REGION Network 18: Robot1Grip Code
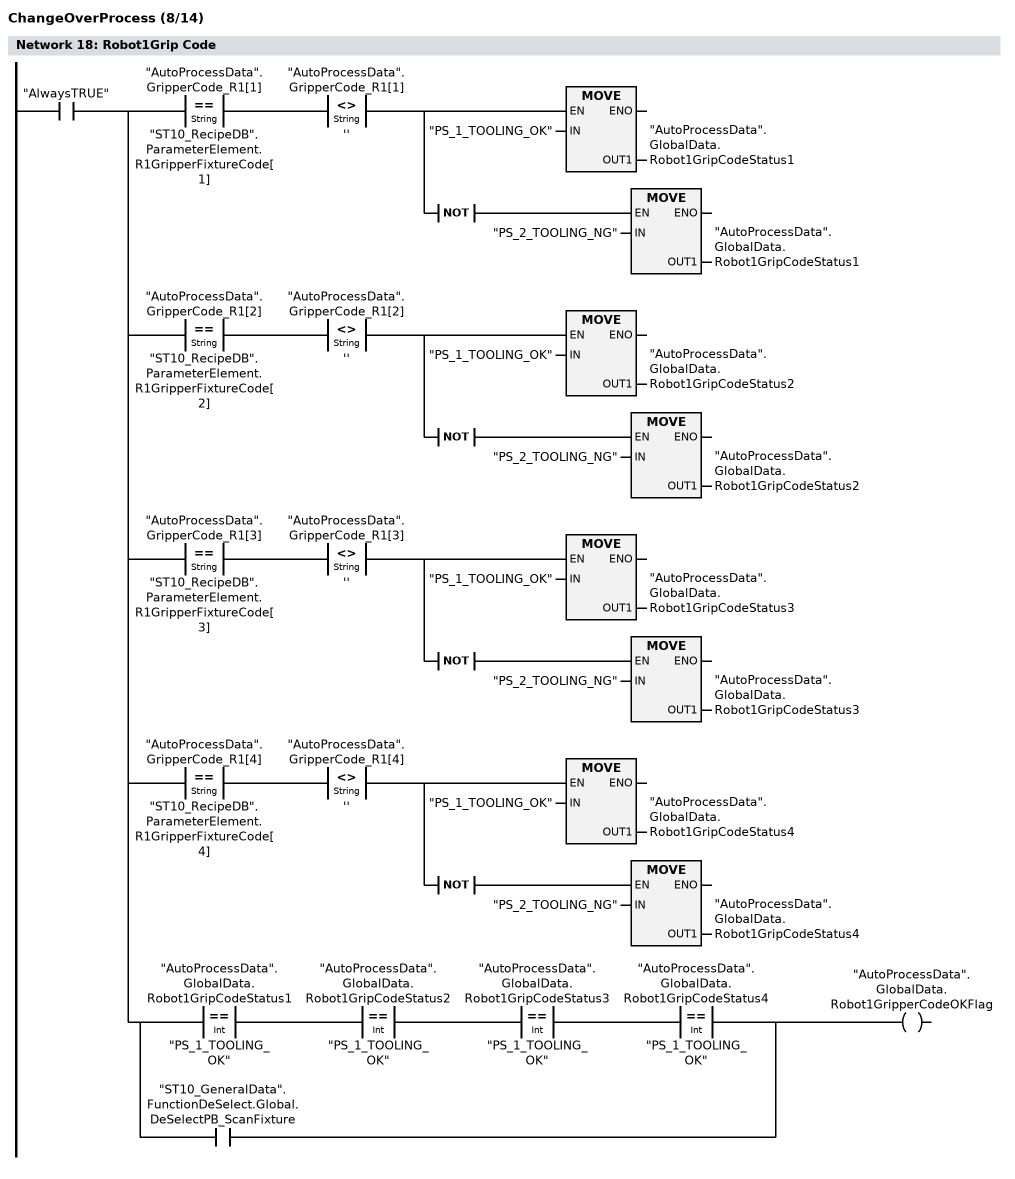
   RUNG wire#powerrail
      Contact( "AlwaysTRUE" )
      wire#w1
      { S7_Templates := "SrcType := String" } EQ_Contact(in1 := "AutoProcessData".GripperCode_R1[1], in2 := "ST10_RecipeDB".ParameterElement.R1GripperFixtureCode[1])
      { S7_Templates := "SrcType := String" } NE_Contact(in1 := "AutoProcessData".GripperCode_R1[1], in2 := '')
      wire#w2
      Move(in := "PS_1_TOOLING_OK", out1 => "AutoProcessData".GlobalData.Robot1GripCodeStatus1)
   END_RUNG
   RUNG wire#w2
      Not()
      Move(in := "PS_2_TOOLING_NG", out1 => "AutoProcessData".GlobalData.Robot1GripCodeStatus1)
   END_RUNG
   RUNG wire#w1
      { S7_Templates := "SrcType := String" } EQ_Contact(in1 := "AutoProcessData".GripperCode_R1[2], in2 := "ST10_RecipeDB".ParameterElement.R1GripperFixtureCode[2])
      { S7_Templates := "SrcType := String" } NE_Contact(in1 := "AutoProcessData".GripperCode_R1[2], in2 := '')
      wire#w3
      Move(in := "PS_1_TOOLING_OK", out1 => "AutoProcessData".GlobalData.Robot1GripCodeStatus2)
   END_RUNG
   RUNG wire#w3
      Not()
      Move(in := "PS_2_TOOLING_NG", out1 => "AutoProcessData".GlobalData.Robot1GripCodeStatus2)
   END_RUNG
   RUNG wire#w1
      { S7_Templates := "SrcType := String" } EQ_Contact(in1 := "AutoProcessData".GripperCode_R1[3], in2 := "ST10_RecipeDB".ParameterElement.R1GripperFixtureCode[3])
      { S7_Templates := "SrcType := String" } NE_Contact(in1 := "AutoProcessData".GripperCode_R1[3], in2 := '')
      wire#w4
      Move(in := "PS_1_TOOLING_OK", out1 => "AutoProcessData".GlobalData.Robot1GripCodeStatus3)
   END_RUNG
   RUNG wire#w4
      Not()
      Move(in := "PS_2_TOOLING_NG", out1 => "AutoProcessData".GlobalData.Robot1GripCodeStatus3)
   END_RUNG
   RUNG wire#w1
      { S7_Templates := "SrcType := String" } EQ_Contact(in1 := "AutoProcessData".GripperCode_R1[4], in2 := "ST10_RecipeDB".ParameterElement.R1GripperFixtureCode[4])
      { S7_Templates := "SrcType := String" } NE_Contact(in1 := "AutoProcessData".GripperCode_R1[4], in2 := '')
      wire#w5
      Move(in := "PS_1_TOOLING_OK", out1 => "AutoProcessData".GlobalData.Robot1GripCodeStatus4)
   END_RUNG
   RUNG wire#w5
      Not()
      Move(in := "PS_2_TOOLING_NG", out1 => "AutoProcessData".GlobalData.Robot1GripCodeStatus4)
   END_RUNG
   RUNG wire#w1
      { S7_Templates := "SrcType := Int" } EQ_Contact(in1 := "AutoProcessData".GlobalData.Robot1GripCodeStatus1, in2 := "PS_1_TOOLING_OK")
      { S7_Templates := "SrcType := Int" } EQ_Contact(in1 := "AutoProcessData".GlobalData.Robot1GripCodeStatus2, in2 := "PS_1_TOOLING_OK")
      { S7_Templates := "SrcType := Int" } EQ_Contact(in1 := "AutoProcessData".GlobalData.Robot1GripCodeStatus3, in2 := "PS_1_TOOLING_OK")
      { S7_Templates := "SrcType := Int" } EQ_Contact(in1 := "AutoProcessData".GlobalData.Robot1GripCodeStatus4, in2 := "PS_1_TOOLING_OK")
      wire#w6
      Coil( "AutoProcessData".GlobalData.Robot1GripperCodeOKFlag )
   END_RUNG
   RUNG wire#w1
      Contact( "ST10_GeneralData".FunctionDeSelect.Global.DeSelectPB_ScanFixture )
   END_RUNG wire#w6
   // the same network as SCL:
   #_w1 := "AlwaysTRUE" AND ("AutoProcessData".GripperCode_R1[1] = "ST10_RecipeDB".ParameterElement.R1GripperFixtureCode[1]) AND ("AutoProcessData".GripperCode_R1[1] <> '');
   IF #_w1 THEN "AutoProcessData".GlobalData.Robot1GripCodeStatus1 := "PS_1_TOOLING_OK"; END_IF;
   IF NOT #_w1 THEN "AutoProcessData".GlobalData.Robot1GripCodeStatus1 := "PS_2_TOOLING_NG"; END_IF;
   #_w2 := "AlwaysTRUE" AND ("AutoProcessData".GripperCode_R1[2] = "ST10_RecipeDB".ParameterElement.R1GripperFixtureCode[2]) AND ("AutoProcessData".GripperCode_R1[2] <> '');
   IF #_w2 THEN "AutoProcessData".GlobalData.Robot1GripCodeStatus2 := "PS_1_TOOLING_OK"; END_IF;
   IF NOT #_w2 THEN "AutoProcessData".GlobalData.Robot1GripCodeStatus2 := "PS_2_TOOLING_NG"; END_IF;
   #_w3 := "AlwaysTRUE" AND ("AutoProcessData".GripperCode_R1[3] = "ST10_RecipeDB".ParameterElement.R1GripperFixtureCode[3]) AND ("AutoProcessData".GripperCode_R1[3] <> '');
   IF #_w3 THEN "AutoProcessData".GlobalData.Robot1GripCodeStatus3 := "PS_1_TOOLING_OK"; END_IF;
   IF NOT #_w3 THEN "AutoProcessData".GlobalData.Robot1GripCodeStatus3 := "PS_2_TOOLING_NG"; END_IF;
   #_w4 := "AlwaysTRUE" AND ("AutoProcessData".GripperCode_R1[4] = "ST10_RecipeDB".ParameterElement.R1GripperFixtureCode[4]) AND ("AutoProcessData".GripperCode_R1[4] <> '');
   IF #_w4 THEN "AutoProcessData".GlobalData.Robot1GripCodeStatus4 := "PS_1_TOOLING_OK"; END_IF;
   IF NOT #_w4 THEN "AutoProcessData".GlobalData.Robot1GripCodeStatus4 := "PS_2_TOOLING_NG"; END_IF;
   "AutoProcessData".GlobalData.Robot1GripperCodeOKFlag := "AlwaysTRUE" AND ((("AutoProcessData".GlobalData.Robot1GripCodeStatus1 = "PS_1_TOOLING_OK") AND ("AutoProcessData".GlobalData.Robot1GripCodeStatus2 = "PS_1_TOOLING_OK") AND ("AutoProcessData".GlobalData.Robot1GripCodeStatus3 = "PS_1_TOOLING_OK") AND ("AutoProcessData".GlobalData.Robot1GripCodeStatus4 = "PS_1_TOOLING_OK")) OR "ST10_GeneralData".FunctionDeSelect.Global.DeSelectPB_ScanFixture);
END_REGION

REGION Network 19: Robot2Grip Code
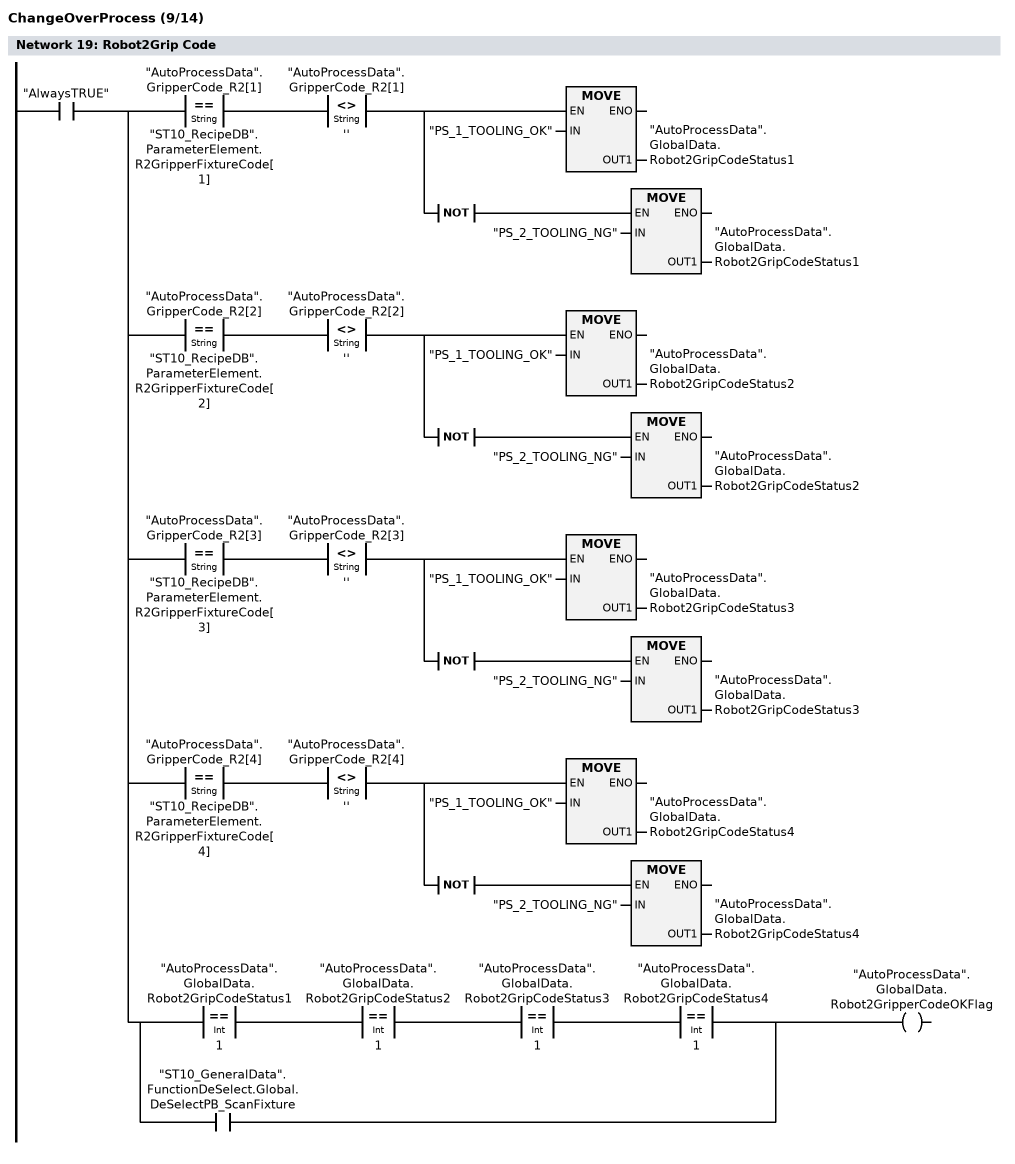
   RUNG wire#powerrail
      Contact( "AlwaysTRUE" )
      wire#w1
      { S7_Templates := "SrcType := String" } EQ_Contact(in1 := "AutoProcessData".GripperCode_R2[1], in2 := "ST10_RecipeDB".ParameterElement.R2GripperFixtureCode[1])
      { S7_Templates := "SrcType := String" } NE_Contact(in1 := "AutoProcessData".GripperCode_R2[1], in2 := '')
      wire#w2
      Move(in := "PS_1_TOOLING_OK", out1 => "AutoProcessData".GlobalData.Robot2GripCodeStatus1)
   END_RUNG
   RUNG wire#w2
      Not()
      Move(in := "PS_2_TOOLING_NG", out1 => "AutoProcessData".GlobalData.Robot2GripCodeStatus1)
   END_RUNG
   RUNG wire#w1
      { S7_Templates := "SrcType := String" } EQ_Contact(in1 := "AutoProcessData".GripperCode_R2[2], in2 := "ST10_RecipeDB".ParameterElement.R2GripperFixtureCode[2])
      { S7_Templates := "SrcType := String" } NE_Contact(in1 := "AutoProcessData".GripperCode_R2[2], in2 := '')
      wire#w3
      Move(in := "PS_1_TOOLING_OK", out1 => "AutoProcessData".GlobalData.Robot2GripCodeStatus2)
   END_RUNG
   RUNG wire#w3
      Not()
      Move(in := "PS_2_TOOLING_NG", out1 => "AutoProcessData".GlobalData.Robot2GripCodeStatus2)
   END_RUNG
   RUNG wire#w1
      { S7_Templates := "SrcType := String" } EQ_Contact(in1 := "AutoProcessData".GripperCode_R2[3], in2 := "ST10_RecipeDB".ParameterElement.R2GripperFixtureCode[3])
      { S7_Templates := "SrcType := String" } NE_Contact(in1 := "AutoProcessData".GripperCode_R2[3], in2 := '')
      wire#w4
      Move(in := "PS_1_TOOLING_OK", out1 => "AutoProcessData".GlobalData.Robot2GripCodeStatus3)
   END_RUNG
   RUNG wire#w4
      Not()
      Move(in := "PS_2_TOOLING_NG", out1 => "AutoProcessData".GlobalData.Robot2GripCodeStatus3)
   END_RUNG
   RUNG wire#w1
      { S7_Templates := "SrcType := String" } EQ_Contact(in1 := "AutoProcessData".GripperCode_R2[4], in2 := "ST10_RecipeDB".ParameterElement.R2GripperFixtureCode[4])
      { S7_Templates := "SrcType := String" } NE_Contact(in1 := "AutoProcessData".GripperCode_R2[4], in2 := '')
      wire#w5
      Move(in := "PS_1_TOOLING_OK", out1 => "AutoProcessData".GlobalData.Robot2GripCodeStatus4)
   END_RUNG
   RUNG wire#w5
      Not()
      Move(in := "PS_2_TOOLING_NG", out1 => "AutoProcessData".GlobalData.Robot2GripCodeStatus4)
   END_RUNG
   RUNG wire#w1
      { S7_Templates := "SrcType := Int" } EQ_Contact(in1 := "AutoProcessData".GlobalData.Robot2GripCodeStatus1, in2 := 1)
      { S7_Templates := "SrcType := Int" } EQ_Contact(in1 := "AutoProcessData".GlobalData.Robot2GripCodeStatus2, in2 := 1)
      { S7_Templates := "SrcType := Int" } EQ_Contact(in1 := "AutoProcessData".GlobalData.Robot2GripCodeStatus3, in2 := 1)
      { S7_Templates := "SrcType := Int" } EQ_Contact(in1 := "AutoProcessData".GlobalData.Robot2GripCodeStatus4, in2 := 1)
      wire#w6
      Coil( "AutoProcessData".GlobalData.Robot2GripperCodeOKFlag )
   END_RUNG
   RUNG wire#w1
      Contact( "ST10_GeneralData".FunctionDeSelect.Global.DeSelectPB_ScanFixture )
   END_RUNG wire#w6
   // the same network as SCL:
   #_w1 := "AlwaysTRUE" AND ("AutoProcessData".GripperCode_R2[1] = "ST10_RecipeDB".ParameterElement.R2GripperFixtureCode[1]) AND ("AutoProcessData".GripperCode_R2[1] <> '');
   IF #_w1 THEN "AutoProcessData".GlobalData.Robot2GripCodeStatus1 := "PS_1_TOOLING_OK"; END_IF;
   IF NOT #_w1 THEN "AutoProcessData".GlobalData.Robot2GripCodeStatus1 := "PS_2_TOOLING_NG"; END_IF;
   #_w2 := "AlwaysTRUE" AND ("AutoProcessData".GripperCode_R2[2] = "ST10_RecipeDB".ParameterElement.R2GripperFixtureCode[2]) AND ("AutoProcessData".GripperCode_R2[2] <> '');
   IF #_w2 THEN "AutoProcessData".GlobalData.Robot2GripCodeStatus2 := "PS_1_TOOLING_OK"; END_IF;
   IF NOT #_w2 THEN "AutoProcessData".GlobalData.Robot2GripCodeStatus2 := "PS_2_TOOLING_NG"; END_IF;
   #_w3 := "AlwaysTRUE" AND ("AutoProcessData".GripperCode_R2[3] = "ST10_RecipeDB".ParameterElement.R2GripperFixtureCode[3]) AND ("AutoProcessData".GripperCode_R2[3] <> '');
   IF #_w3 THEN "AutoProcessData".GlobalData.Robot2GripCodeStatus3 := "PS_1_TOOLING_OK"; END_IF;
   IF NOT #_w3 THEN "AutoProcessData".GlobalData.Robot2GripCodeStatus3 := "PS_2_TOOLING_NG"; END_IF;
   #_w4 := "AlwaysTRUE" AND ("AutoProcessData".GripperCode_R2[4] = "ST10_RecipeDB".ParameterElement.R2GripperFixtureCode[4]) AND ("AutoProcessData".GripperCode_R2[4] <> '');
   IF #_w4 THEN "AutoProcessData".GlobalData.Robot2GripCodeStatus4 := "PS_1_TOOLING_OK"; END_IF;
   IF NOT #_w4 THEN "AutoProcessData".GlobalData.Robot2GripCodeStatus4 := "PS_2_TOOLING_NG"; END_IF;
   "AutoProcessData".GlobalData.Robot2GripperCodeOKFlag := "AlwaysTRUE" AND ((("AutoProcessData".GlobalData.Robot2GripCodeStatus1 = 1) AND ("AutoProcessData".GlobalData.Robot2GripCodeStatus2 = 1) AND ("AutoProcessData".GlobalData.Robot2GripCodeStatus3 = 1) AND ("AutoProcessData".GlobalData.Robot2GripCodeStatus4 = 1)) OR "ST10_GeneralData".FunctionDeSelect.Global.DeSelectPB_ScanFixture);
END_REGION

REGION Network 20: Robot3Grip Code
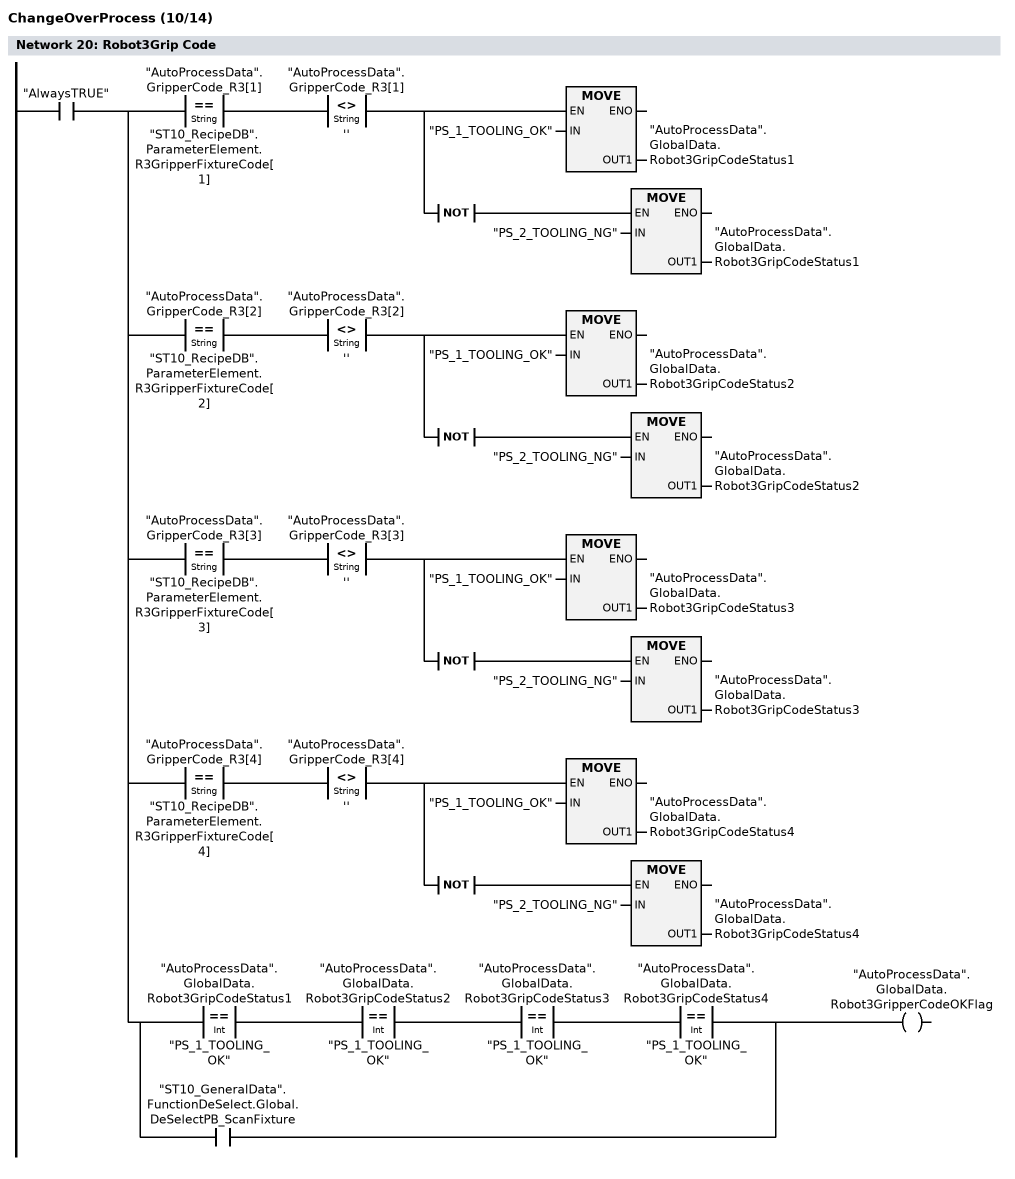
   RUNG wire#powerrail
      Contact( "AlwaysTRUE" )
      wire#w1
      { S7_Templates := "SrcType := String" } EQ_Contact(in1 := "AutoProcessData".GripperCode_R3[1], in2 := "ST10_RecipeDB".ParameterElement.R3GripperFixtureCode[1])
      { S7_Templates := "SrcType := String" } NE_Contact(in1 := "AutoProcessData".GripperCode_R3[1], in2 := '')
      wire#w2
      Move(in := "PS_1_TOOLING_OK", out1 => "AutoProcessData".GlobalData.Robot3GripCodeStatus1)
   END_RUNG
   RUNG wire#w2
      Not()
      Move(in := "PS_2_TOOLING_NG", out1 => "AutoProcessData".GlobalData.Robot3GripCodeStatus1)
   END_RUNG
   RUNG wire#w1
      { S7_Templates := "SrcType := String" } EQ_Contact(in1 := "AutoProcessData".GripperCode_R3[2], in2 := "ST10_RecipeDB".ParameterElement.R3GripperFixtureCode[2])
      { S7_Templates := "SrcType := String" } NE_Contact(in1 := "AutoProcessData".GripperCode_R3[2], in2 := '')
      wire#w3
      Move(in := "PS_1_TOOLING_OK", out1 => "AutoProcessData".GlobalData.Robot3GripCodeStatus2)
   END_RUNG
   RUNG wire#w3
      Not()
      Move(in := "PS_2_TOOLING_NG", out1 => "AutoProcessData".GlobalData.Robot3GripCodeStatus2)
   END_RUNG
   RUNG wire#w1
      { S7_Templates := "SrcType := String" } EQ_Contact(in1 := "AutoProcessData".GripperCode_R3[3], in2 := "ST10_RecipeDB".ParameterElement.R3GripperFixtureCode[3])
      { S7_Templates := "SrcType := String" } NE_Contact(in1 := "AutoProcessData".GripperCode_R3[3], in2 := '')
      wire#w4
      Move(in := "PS_1_TOOLING_OK", out1 => "AutoProcessData".GlobalData.Robot3GripCodeStatus3)
   END_RUNG
   RUNG wire#w4
      Not()
      Move(in := "PS_2_TOOLING_NG", out1 => "AutoProcessData".GlobalData.Robot3GripCodeStatus3)
   END_RUNG
   RUNG wire#w1
      { S7_Templates := "SrcType := String" } EQ_Contact(in1 := "AutoProcessData".GripperCode_R3[4], in2 := "ST10_RecipeDB".ParameterElement.R3GripperFixtureCode[4])
      { S7_Templates := "SrcType := String" } NE_Contact(in1 := "AutoProcessData".GripperCode_R3[4], in2 := '')
      wire#w5
      Move(in := "PS_1_TOOLING_OK", out1 => "AutoProcessData".GlobalData.Robot3GripCodeStatus4)
   END_RUNG
   RUNG wire#w5
      Not()
      Move(in := "PS_2_TOOLING_NG", out1 => "AutoProcessData".GlobalData.Robot3GripCodeStatus4)
   END_RUNG
   RUNG wire#w1
      { S7_Templates := "SrcType := Int" } EQ_Contact(in1 := "AutoProcessData".GlobalData.Robot3GripCodeStatus1, in2 := "PS_1_TOOLING_OK")
      { S7_Templates := "SrcType := Int" } EQ_Contact(in1 := "AutoProcessData".GlobalData.Robot3GripCodeStatus2, in2 := "PS_1_TOOLING_OK")
      { S7_Templates := "SrcType := Int" } EQ_Contact(in1 := "AutoProcessData".GlobalData.Robot3GripCodeStatus3, in2 := "PS_1_TOOLING_OK")
      { S7_Templates := "SrcType := Int" } EQ_Contact(in1 := "AutoProcessData".GlobalData.Robot3GripCodeStatus4, in2 := "PS_1_TOOLING_OK")
      wire#w6
      Coil( "AutoProcessData".GlobalData.Robot3GripperCodeOKFlag )
   END_RUNG
   RUNG wire#w1
      Contact( "ST10_GeneralData".FunctionDeSelect.Global.DeSelectPB_ScanFixture )
   END_RUNG wire#w6
   // the same network as SCL:
   #_w1 := "AlwaysTRUE" AND ("AutoProcessData".GripperCode_R3[1] = "ST10_RecipeDB".ParameterElement.R3GripperFixtureCode[1]) AND ("AutoProcessData".GripperCode_R3[1] <> '');
   IF #_w1 THEN "AutoProcessData".GlobalData.Robot3GripCodeStatus1 := "PS_1_TOOLING_OK"; END_IF;
   IF NOT #_w1 THEN "AutoProcessData".GlobalData.Robot3GripCodeStatus1 := "PS_2_TOOLING_NG"; END_IF;
   #_w2 := "AlwaysTRUE" AND ("AutoProcessData".GripperCode_R3[2] = "ST10_RecipeDB".ParameterElement.R3GripperFixtureCode[2]) AND ("AutoProcessData".GripperCode_R3[2] <> '');
   IF #_w2 THEN "AutoProcessData".GlobalData.Robot3GripCodeStatus2 := "PS_1_TOOLING_OK"; END_IF;
   IF NOT #_w2 THEN "AutoProcessData".GlobalData.Robot3GripCodeStatus2 := "PS_2_TOOLING_NG"; END_IF;
   #_w3 := "AlwaysTRUE" AND ("AutoProcessData".GripperCode_R3[3] = "ST10_RecipeDB".ParameterElement.R3GripperFixtureCode[3]) AND ("AutoProcessData".GripperCode_R3[3] <> '');
   IF #_w3 THEN "AutoProcessData".GlobalData.Robot3GripCodeStatus3 := "PS_1_TOOLING_OK"; END_IF;
   IF NOT #_w3 THEN "AutoProcessData".GlobalData.Robot3GripCodeStatus3 := "PS_2_TOOLING_NG"; END_IF;
   #_w4 := "AlwaysTRUE" AND ("AutoProcessData".GripperCode_R3[4] = "ST10_RecipeDB".ParameterElement.R3GripperFixtureCode[4]) AND ("AutoProcessData".GripperCode_R3[4] <> '');
   IF #_w4 THEN "AutoProcessData".GlobalData.Robot3GripCodeStatus4 := "PS_1_TOOLING_OK"; END_IF;
   IF NOT #_w4 THEN "AutoProcessData".GlobalData.Robot3GripCodeStatus4 := "PS_2_TOOLING_NG"; END_IF;
   "AutoProcessData".GlobalData.Robot3GripperCodeOKFlag := "AlwaysTRUE" AND ((("AutoProcessData".GlobalData.Robot3GripCodeStatus1 = "PS_1_TOOLING_OK") AND ("AutoProcessData".GlobalData.Robot3GripCodeStatus2 = "PS_1_TOOLING_OK") AND ("AutoProcessData".GlobalData.Robot3GripCodeStatus3 = "PS_1_TOOLING_OK") AND ("AutoProcessData".GlobalData.Robot3GripCodeStatus4 = "PS_1_TOOLING_OK")) OR "ST10_GeneralData".FunctionDeSelect.Global.DeSelectPB_ScanFixture);
END_REGION

REGION Network 21: A1 Fixture Code
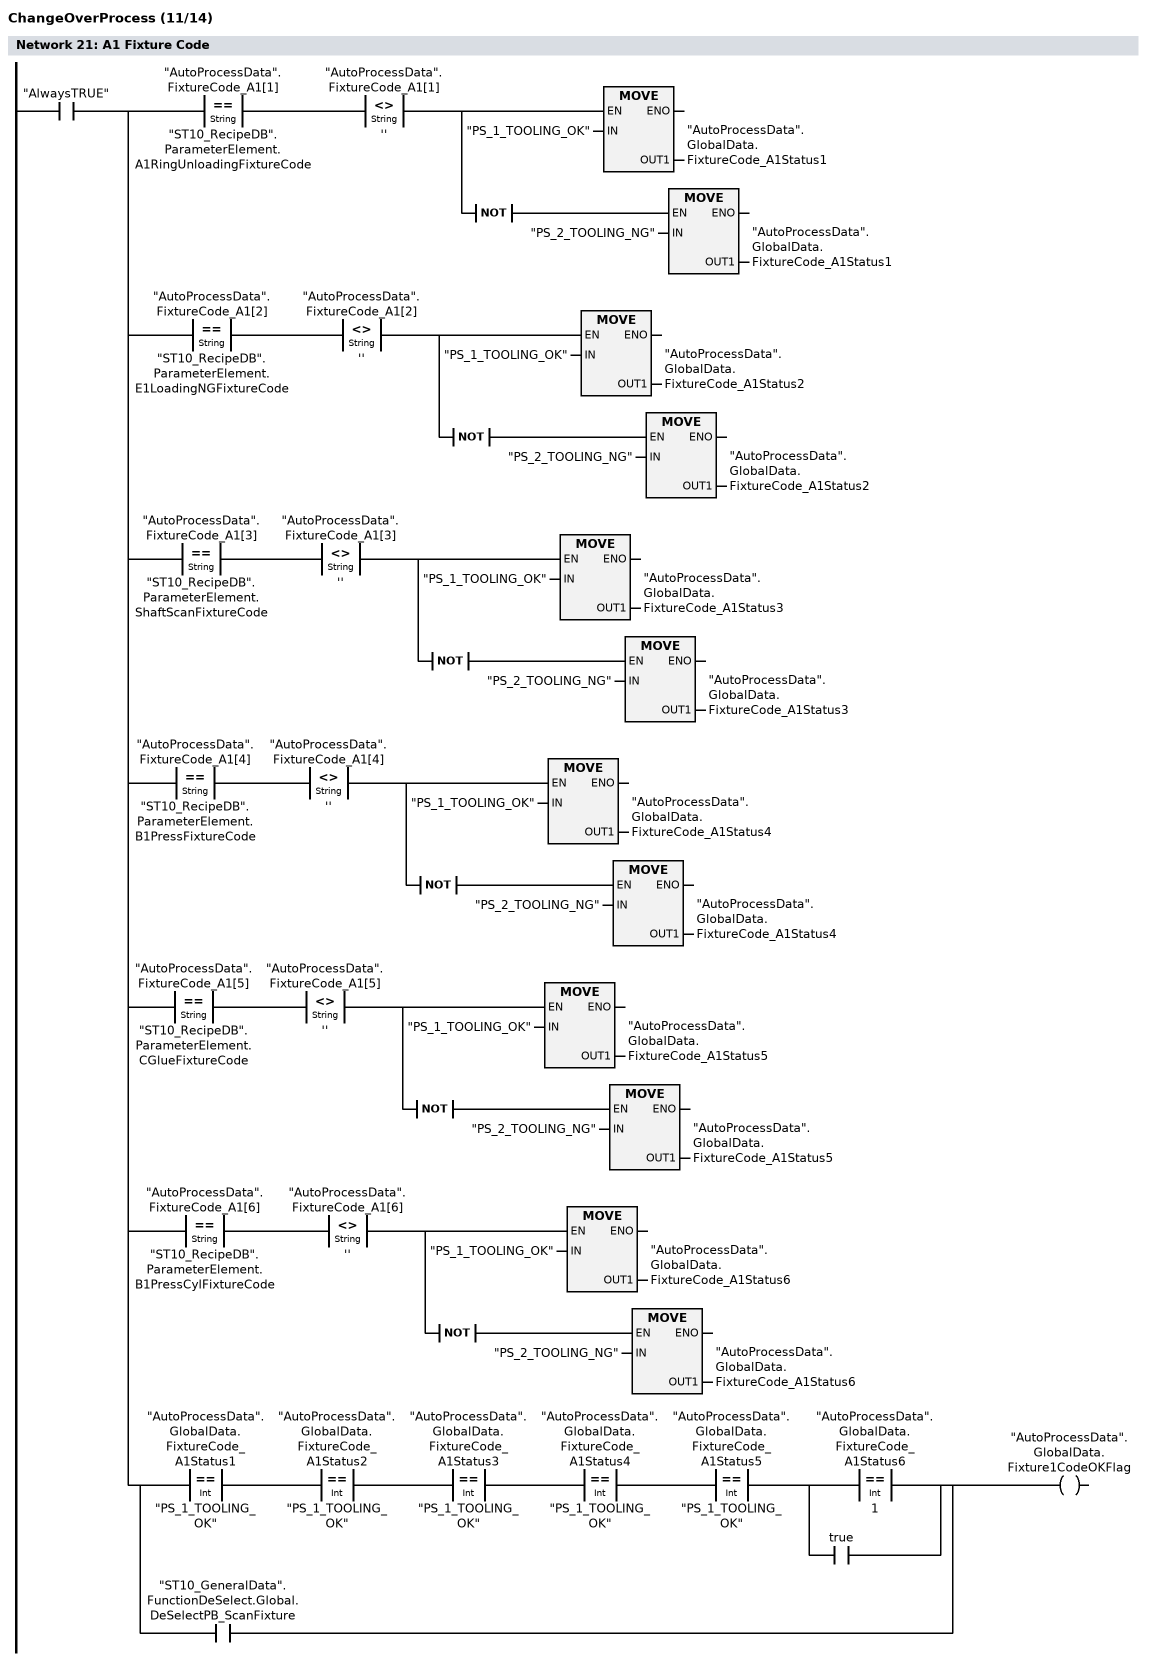
   RUNG wire#powerrail
      Contact( "AlwaysTRUE" )
      wire#w1
      { S7_Templates := "SrcType := String" } EQ_Contact(in1 := "AutoProcessData".FixtureCode_A1[1], in2 := "ST10_RecipeDB".ParameterElement.A1RingUnloadingFixtureCode)
      { S7_Templates := "SrcType := String" } NE_Contact(in1 := "AutoProcessData".FixtureCode_A1[1], in2 := '')
      wire#w2
      Move(in := "PS_1_TOOLING_OK", out1 => "AutoProcessData".GlobalData.FixtureCode_A1Status1)
   END_RUNG
   RUNG wire#w2
      Not()
      Move(in := "PS_2_TOOLING_NG", out1 => "AutoProcessData".GlobalData.FixtureCode_A1Status1)
   END_RUNG
   RUNG wire#w1
      { S7_Templates := "SrcType := String" } EQ_Contact(in1 := "AutoProcessData".FixtureCode_A1[2], in2 := "ST10_RecipeDB".ParameterElement.E1LoadingNGFixtureCode)
      { S7_Templates := "SrcType := String" } NE_Contact(in1 := "AutoProcessData".FixtureCode_A1[2], in2 := '')
      wire#w3
      Move(in := "PS_1_TOOLING_OK", out1 => "AutoProcessData".GlobalData.FixtureCode_A1Status2)
   END_RUNG
   RUNG wire#w3
      Not()
      Move(in := "PS_2_TOOLING_NG", out1 => "AutoProcessData".GlobalData.FixtureCode_A1Status2)
   END_RUNG
   RUNG wire#w1
      { S7_Templates := "SrcType := String" } EQ_Contact(in1 := "AutoProcessData".FixtureCode_A1[3], in2 := "ST10_RecipeDB".ParameterElement.ShaftScanFixtureCode)
      { S7_Templates := "SrcType := String" } NE_Contact(in1 := "AutoProcessData".FixtureCode_A1[3], in2 := '')
      wire#w4
      Move(in := "PS_1_TOOLING_OK", out1 => "AutoProcessData".GlobalData.FixtureCode_A1Status3)
   END_RUNG
   RUNG wire#w4
      Not()
      Move(in := "PS_2_TOOLING_NG", out1 => "AutoProcessData".GlobalData.FixtureCode_A1Status3)
   END_RUNG
   RUNG wire#w1
      { S7_Templates := "SrcType := String" } EQ_Contact(in1 := "AutoProcessData".FixtureCode_A1[4], in2 := "ST10_RecipeDB".ParameterElement.B1PressFixtureCode)
      { S7_Templates := "SrcType := String" } NE_Contact(in1 := "AutoProcessData".FixtureCode_A1[4], in2 := '')
      wire#w5
      Move(in := "PS_1_TOOLING_OK", out1 => "AutoProcessData".GlobalData.FixtureCode_A1Status4)
   END_RUNG
   RUNG wire#w5
      Not()
      Move(in := "PS_2_TOOLING_NG", out1 => "AutoProcessData".GlobalData.FixtureCode_A1Status4)
   END_RUNG
   RUNG wire#w1
      { S7_Templates := "SrcType := String" } EQ_Contact(in1 := "AutoProcessData".FixtureCode_A1[5], in2 := "ST10_RecipeDB".ParameterElement.CGlueFixtureCode)
      { S7_Templates := "SrcType := String" } NE_Contact(in1 := "AutoProcessData".FixtureCode_A1[5], in2 := '')
      wire#w6
      Move(in := "PS_1_TOOLING_OK", out1 => "AutoProcessData".GlobalData.FixtureCode_A1Status5)
   END_RUNG
   RUNG wire#w6
      Not()
      Move(in := "PS_2_TOOLING_NG", out1 => "AutoProcessData".GlobalData.FixtureCode_A1Status5)
   END_RUNG
   RUNG wire#w1
      { S7_Templates := "SrcType := String" } EQ_Contact(in1 := "AutoProcessData".FixtureCode_A1[6], in2 := "ST10_RecipeDB".ParameterElement.B1PressCylFixtureCode)
      { S7_Templates := "SrcType := String" } NE_Contact(in1 := "AutoProcessData".FixtureCode_A1[6], in2 := '')
      wire#w7
      Move(in := "PS_1_TOOLING_OK", out1 => "AutoProcessData".GlobalData.FixtureCode_A1Status6)
   END_RUNG
   RUNG wire#w7
      Not()
      Move(in := "PS_2_TOOLING_NG", out1 => "AutoProcessData".GlobalData.FixtureCode_A1Status6)
   END_RUNG
   RUNG wire#w1
      { S7_Templates := "SrcType := Int" } EQ_Contact(in1 := "AutoProcessData".GlobalData.FixtureCode_A1Status1, in2 := "PS_1_TOOLING_OK")
      { S7_Templates := "SrcType := Int" } EQ_Contact(in1 := "AutoProcessData".GlobalData.FixtureCode_A1Status2, in2 := "PS_1_TOOLING_OK")
      { S7_Templates := "SrcType := Int" } EQ_Contact(in1 := "AutoProcessData".GlobalData.FixtureCode_A1Status3, in2 := "PS_1_TOOLING_OK")
      { S7_Templates := "SrcType := Int" } EQ_Contact(in1 := "AutoProcessData".GlobalData.FixtureCode_A1Status4, in2 := "PS_1_TOOLING_OK")
      { S7_Templates := "SrcType := Int" } EQ_Contact(in1 := "AutoProcessData".GlobalData.FixtureCode_A1Status5, in2 := "PS_1_TOOLING_OK")
      wire#w8
      { S7_Templates := "SrcType := Int" } EQ_Contact(in1 := "AutoProcessData".GlobalData.FixtureCode_A1Status6, in2 := 1)
      wire#w9
      Coil( "AutoProcessData".GlobalData.Fixture1CodeOKFlag )
   END_RUNG
   RUNG wire#w8
      Contact( true )
   END_RUNG wire#w9
   RUNG wire#w1
      Contact( "ST10_GeneralData".FunctionDeSelect.Global.DeSelectPB_ScanFixture )
   END_RUNG wire#w9
   // the same network as SCL:
   #_w1 := "AlwaysTRUE" AND ("AutoProcessData".FixtureCode_A1[1] = "ST10_RecipeDB".ParameterElement.A1RingUnloadingFixtureCode) AND ("AutoProcessData".FixtureCode_A1[1] <> '');
   IF #_w1 THEN "AutoProcessData".GlobalData.FixtureCode_A1Status1 := "PS_1_TOOLING_OK"; END_IF;
   IF NOT #_w1 THEN "AutoProcessData".GlobalData.FixtureCode_A1Status1 := "PS_2_TOOLING_NG"; END_IF;
   #_w2 := "AlwaysTRUE" AND ("AutoProcessData".FixtureCode_A1[2] = "ST10_RecipeDB".ParameterElement.E1LoadingNGFixtureCode) AND ("AutoProcessData".FixtureCode_A1[2] <> '');
   IF #_w2 THEN "AutoProcessData".GlobalData.FixtureCode_A1Status2 := "PS_1_TOOLING_OK"; END_IF;
   IF NOT #_w2 THEN "AutoProcessData".GlobalData.FixtureCode_A1Status2 := "PS_2_TOOLING_NG"; END_IF;
   #_w3 := "AlwaysTRUE" AND ("AutoProcessData".FixtureCode_A1[3] = "ST10_RecipeDB".ParameterElement.ShaftScanFixtureCode) AND ("AutoProcessData".FixtureCode_A1[3] <> '');
   IF #_w3 THEN "AutoProcessData".GlobalData.FixtureCode_A1Status3 := "PS_1_TOOLING_OK"; END_IF;
   IF NOT #_w3 THEN "AutoProcessData".GlobalData.FixtureCode_A1Status3 := "PS_2_TOOLING_NG"; END_IF;
   #_w4 := "AlwaysTRUE" AND ("AutoProcessData".FixtureCode_A1[4] = "ST10_RecipeDB".ParameterElement.B1PressFixtureCode) AND ("AutoProcessData".FixtureCode_A1[4] <> '');
   IF #_w4 THEN "AutoProcessData".GlobalData.FixtureCode_A1Status4 := "PS_1_TOOLING_OK"; END_IF;
   IF NOT #_w4 THEN "AutoProcessData".GlobalData.FixtureCode_A1Status4 := "PS_2_TOOLING_NG"; END_IF;
   #_w5 := "AlwaysTRUE" AND ("AutoProcessData".FixtureCode_A1[5] = "ST10_RecipeDB".ParameterElement.CGlueFixtureCode) AND ("AutoProcessData".FixtureCode_A1[5] <> '');
   IF #_w5 THEN "AutoProcessData".GlobalData.FixtureCode_A1Status5 := "PS_1_TOOLING_OK"; END_IF;
   IF NOT #_w5 THEN "AutoProcessData".GlobalData.FixtureCode_A1Status5 := "PS_2_TOOLING_NG"; END_IF;
   #_w6 := "AlwaysTRUE" AND ("AutoProcessData".FixtureCode_A1[6] = "ST10_RecipeDB".ParameterElement.B1PressCylFixtureCode) AND ("AutoProcessData".FixtureCode_A1[6] <> '');
   IF #_w6 THEN "AutoProcessData".GlobalData.FixtureCode_A1Status6 := "PS_1_TOOLING_OK"; END_IF;
   IF NOT #_w6 THEN "AutoProcessData".GlobalData.FixtureCode_A1Status6 := "PS_2_TOOLING_NG"; END_IF;
   "AutoProcessData".GlobalData.Fixture1CodeOKFlag := "AlwaysTRUE" AND ((("AutoProcessData".GlobalData.FixtureCode_A1Status1 = "PS_1_TOOLING_OK") AND ("AutoProcessData".GlobalData.FixtureCode_A1Status2 = "PS_1_TOOLING_OK") AND ("AutoProcessData".GlobalData.FixtureCode_A1Status3 = "PS_1_TOOLING_OK") AND ("AutoProcessData".GlobalData.FixtureCode_A1Status4 = "PS_1_TOOLING_OK") AND ("AutoProcessData".GlobalData.FixtureCode_A1Status5 = "PS_1_TOOLING_OK") AND (("AutoProcessData".GlobalData.FixtureCode_A1Status6 = 1) OR true)) OR "ST10_GeneralData".FunctionDeSelect.Global.DeSelectPB_ScanFixture);
END_REGION

REGION Network 22: A2 Fixture Code
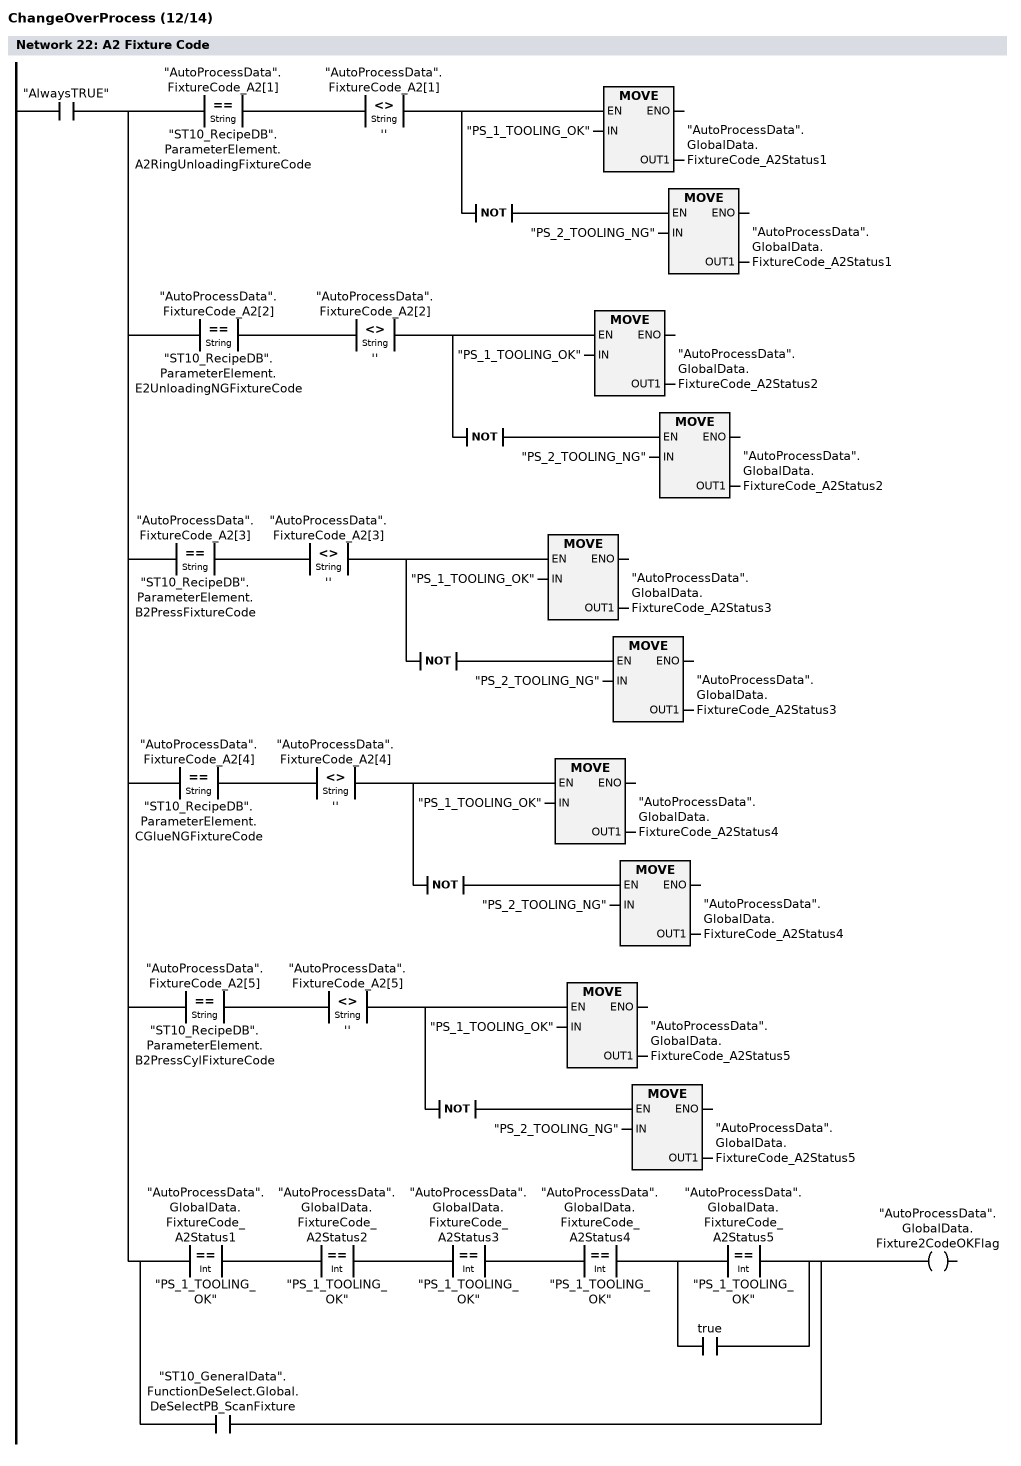
   RUNG wire#powerrail
      Contact( "AlwaysTRUE" )
      wire#w1
      { S7_Templates := "SrcType := String" } EQ_Contact(in1 := "AutoProcessData".FixtureCode_A2[1], in2 := "ST10_RecipeDB".ParameterElement.A2RingUnloadingFixtureCode)
      { S7_Templates := "SrcType := String" } NE_Contact(in1 := "AutoProcessData".FixtureCode_A2[1], in2 := '')
      wire#w2
      Move(in := "PS_1_TOOLING_OK", out1 => "AutoProcessData".GlobalData.FixtureCode_A2Status1)
   END_RUNG
   RUNG wire#w2
      Not()
      Move(in := "PS_2_TOOLING_NG", out1 => "AutoProcessData".GlobalData.FixtureCode_A2Status1)
   END_RUNG
   RUNG wire#w1
      { S7_Templates := "SrcType := String" } EQ_Contact(in1 := "AutoProcessData".FixtureCode_A2[2], in2 := "ST10_RecipeDB".ParameterElement.E2UnloadingNGFixtureCode)
      { S7_Templates := "SrcType := String" } NE_Contact(in1 := "AutoProcessData".FixtureCode_A2[2], in2 := '')
      wire#w3
      Move(in := "PS_1_TOOLING_OK", out1 => "AutoProcessData".GlobalData.FixtureCode_A2Status2)
   END_RUNG
   RUNG wire#w3
      Not()
      Move(in := "PS_2_TOOLING_NG", out1 => "AutoProcessData".GlobalData.FixtureCode_A2Status2)
   END_RUNG
   RUNG wire#w1
      { S7_Templates := "SrcType := String" } EQ_Contact(in1 := "AutoProcessData".FixtureCode_A2[3], in2 := "ST10_RecipeDB".ParameterElement.B2PressFixtureCode)
      { S7_Templates := "SrcType := String" } NE_Contact(in1 := "AutoProcessData".FixtureCode_A2[3], in2 := '')
      wire#w4
      Move(in := "PS_1_TOOLING_OK", out1 => "AutoProcessData".GlobalData.FixtureCode_A2Status3)
   END_RUNG
   RUNG wire#w4
      Not()
      Move(in := "PS_2_TOOLING_NG", out1 => "AutoProcessData".GlobalData.FixtureCode_A2Status3)
   END_RUNG
   RUNG wire#w1
      { S7_Templates := "SrcType := String" } EQ_Contact(in1 := "AutoProcessData".FixtureCode_A2[4], in2 := "ST10_RecipeDB".ParameterElement.CGlueNGFixtureCode)
      { S7_Templates := "SrcType := String" } NE_Contact(in1 := "AutoProcessData".FixtureCode_A2[4], in2 := '')
      wire#w5
      Move(in := "PS_1_TOOLING_OK", out1 => "AutoProcessData".GlobalData.FixtureCode_A2Status4)
   END_RUNG
   RUNG wire#w5
      Not()
      Move(in := "PS_2_TOOLING_NG", out1 => "AutoProcessData".GlobalData.FixtureCode_A2Status4)
   END_RUNG
   RUNG wire#w1
      { S7_Templates := "SrcType := String" } EQ_Contact(in1 := "AutoProcessData".FixtureCode_A2[5], in2 := "ST10_RecipeDB".ParameterElement.B2PressCylFixtureCode)
      { S7_Templates := "SrcType := String" } NE_Contact(in1 := "AutoProcessData".FixtureCode_A2[5], in2 := '')
      wire#w6
      Move(in := "PS_1_TOOLING_OK", out1 => "AutoProcessData".GlobalData.FixtureCode_A2Status5)
   END_RUNG
   RUNG wire#w6
      Not()
      Move(in := "PS_2_TOOLING_NG", out1 => "AutoProcessData".GlobalData.FixtureCode_A2Status5)
   END_RUNG
   RUNG wire#w1
      { S7_Templates := "SrcType := Int" } EQ_Contact(in1 := "AutoProcessData".GlobalData.FixtureCode_A2Status1, in2 := "PS_1_TOOLING_OK")
      { S7_Templates := "SrcType := Int" } EQ_Contact(in1 := "AutoProcessData".GlobalData.FixtureCode_A2Status2, in2 := "PS_1_TOOLING_OK")
      { S7_Templates := "SrcType := Int" } EQ_Contact(in1 := "AutoProcessData".GlobalData.FixtureCode_A2Status3, in2 := "PS_1_TOOLING_OK")
      { S7_Templates := "SrcType := Int" } EQ_Contact(in1 := "AutoProcessData".GlobalData.FixtureCode_A2Status4, in2 := "PS_1_TOOLING_OK")
      wire#w7
      { S7_Templates := "SrcType := Int" } EQ_Contact(in1 := "AutoProcessData".GlobalData.FixtureCode_A2Status5, in2 := "PS_1_TOOLING_OK")
      wire#w8
      Coil( "AutoProcessData".GlobalData.Fixture2CodeOKFlag )
   END_RUNG
   RUNG wire#w7
      Contact( true )
   END_RUNG wire#w8
   RUNG wire#w1
      Contact( "ST10_GeneralData".FunctionDeSelect.Global.DeSelectPB_ScanFixture )
   END_RUNG wire#w8
   // the same network as SCL:
   #_w1 := "AlwaysTRUE" AND ("AutoProcessData".FixtureCode_A2[1] = "ST10_RecipeDB".ParameterElement.A2RingUnloadingFixtureCode) AND ("AutoProcessData".FixtureCode_A2[1] <> '');
   IF #_w1 THEN "AutoProcessData".GlobalData.FixtureCode_A2Status1 := "PS_1_TOOLING_OK"; END_IF;
   IF NOT #_w1 THEN "AutoProcessData".GlobalData.FixtureCode_A2Status1 := "PS_2_TOOLING_NG"; END_IF;
   #_w2 := "AlwaysTRUE" AND ("AutoProcessData".FixtureCode_A2[2] = "ST10_RecipeDB".ParameterElement.E2UnloadingNGFixtureCode) AND ("AutoProcessData".FixtureCode_A2[2] <> '');
   IF #_w2 THEN "AutoProcessData".GlobalData.FixtureCode_A2Status2 := "PS_1_TOOLING_OK"; END_IF;
   IF NOT #_w2 THEN "AutoProcessData".GlobalData.FixtureCode_A2Status2 := "PS_2_TOOLING_NG"; END_IF;
   #_w3 := "AlwaysTRUE" AND ("AutoProcessData".FixtureCode_A2[3] = "ST10_RecipeDB".ParameterElement.B2PressFixtureCode) AND ("AutoProcessData".FixtureCode_A2[3] <> '');
   IF #_w3 THEN "AutoProcessData".GlobalData.FixtureCode_A2Status3 := "PS_1_TOOLING_OK"; END_IF;
   IF NOT #_w3 THEN "AutoProcessData".GlobalData.FixtureCode_A2Status3 := "PS_2_TOOLING_NG"; END_IF;
   #_w4 := "AlwaysTRUE" AND ("AutoProcessData".FixtureCode_A2[4] = "ST10_RecipeDB".ParameterElement.CGlueNGFixtureCode) AND ("AutoProcessData".FixtureCode_A2[4] <> '');
   IF #_w4 THEN "AutoProcessData".GlobalData.FixtureCode_A2Status4 := "PS_1_TOOLING_OK"; END_IF;
   IF NOT #_w4 THEN "AutoProcessData".GlobalData.FixtureCode_A2Status4 := "PS_2_TOOLING_NG"; END_IF;
   #_w5 := "AlwaysTRUE" AND ("AutoProcessData".FixtureCode_A2[5] = "ST10_RecipeDB".ParameterElement.B2PressCylFixtureCode) AND ("AutoProcessData".FixtureCode_A2[5] <> '');
   IF #_w5 THEN "AutoProcessData".GlobalData.FixtureCode_A2Status5 := "PS_1_TOOLING_OK"; END_IF;
   IF NOT #_w5 THEN "AutoProcessData".GlobalData.FixtureCode_A2Status5 := "PS_2_TOOLING_NG"; END_IF;
   "AutoProcessData".GlobalData.Fixture2CodeOKFlag := "AlwaysTRUE" AND ((("AutoProcessData".GlobalData.FixtureCode_A2Status1 = "PS_1_TOOLING_OK") AND ("AutoProcessData".GlobalData.FixtureCode_A2Status2 = "PS_1_TOOLING_OK") AND ("AutoProcessData".GlobalData.FixtureCode_A2Status3 = "PS_1_TOOLING_OK") AND ("AutoProcessData".GlobalData.FixtureCode_A2Status4 = "PS_1_TOOLING_OK") AND (("AutoProcessData".GlobalData.FixtureCode_A2Status5 = "PS_1_TOOLING_OK") OR true)) OR "ST10_GeneralData".FunctionDeSelect.Global.DeSelectPB_ScanFixture);
END_REGION

REGION Network 23: ChangeOverFinish
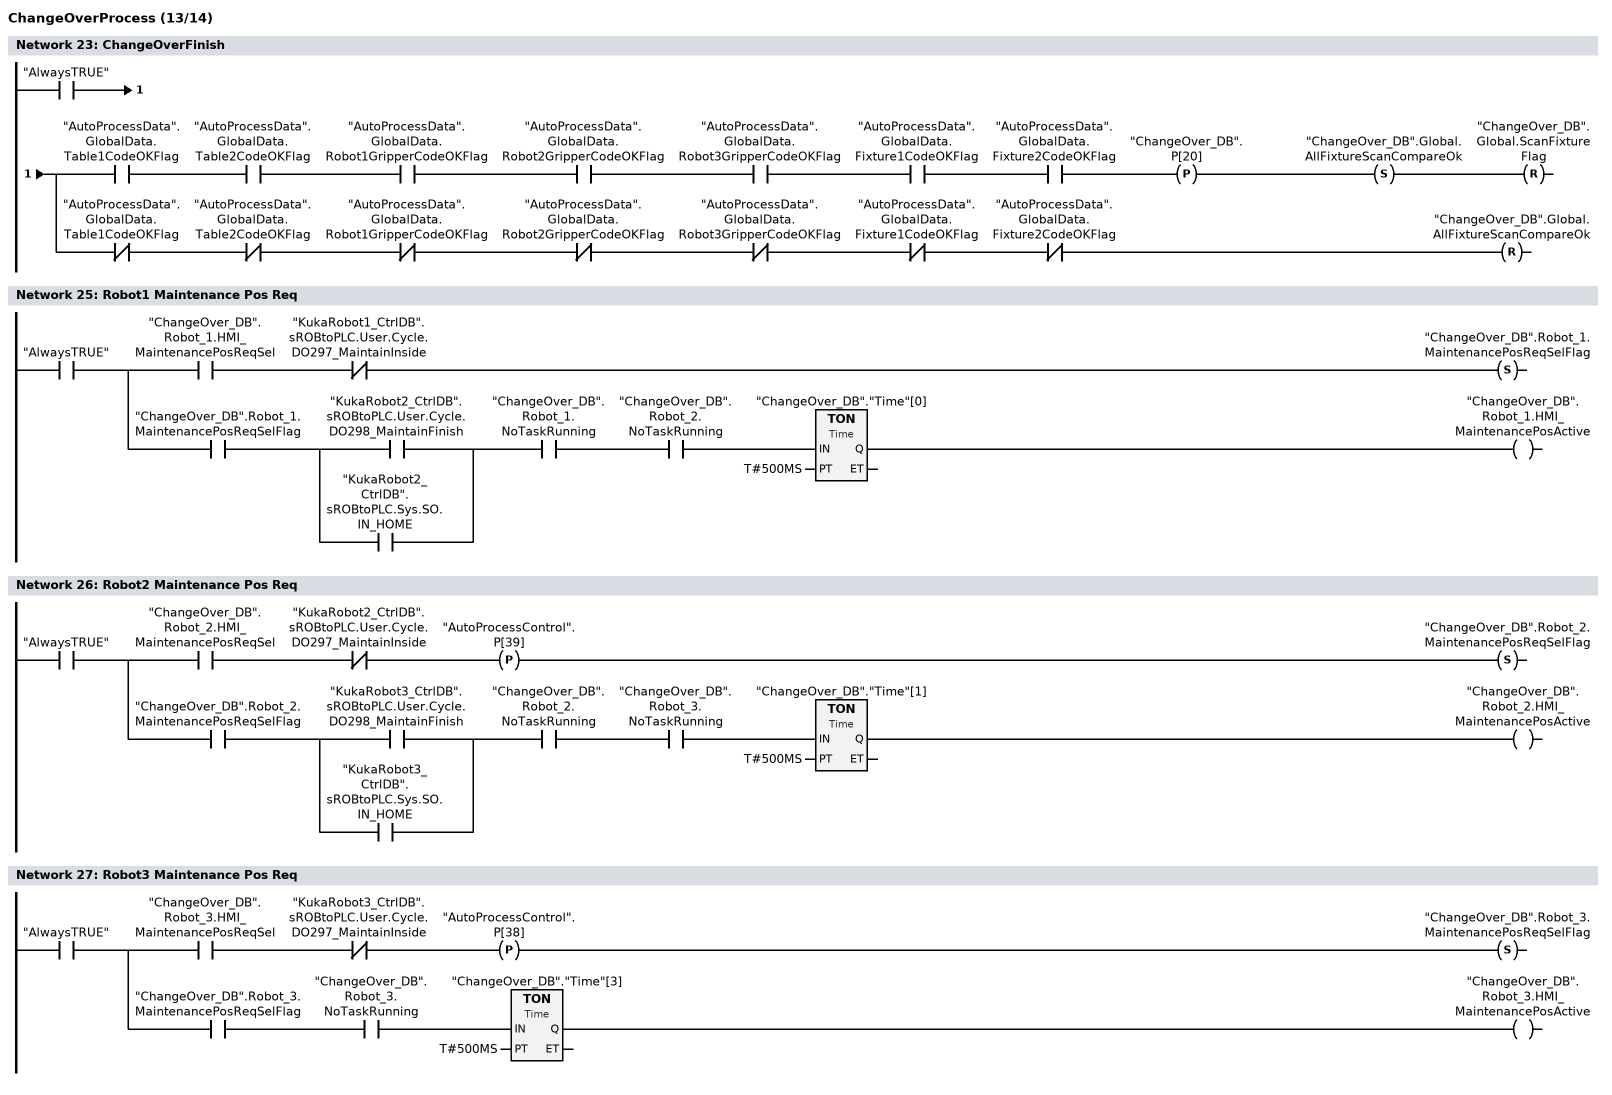
   RUNG wire#powerrail
      Contact( "AlwaysTRUE" )
      wire#w1
      Contact( "AutoProcessData".GlobalData.Table1CodeOKFlag )
      Contact( "AutoProcessData".GlobalData.Table2CodeOKFlag )
      Contact( "AutoProcessData".GlobalData.Robot1GripperCodeOKFlag )
      Contact( "AutoProcessData".GlobalData.Robot2GripperCodeOKFlag )
      Contact( "AutoProcessData".GlobalData.Robot3GripperCodeOKFlag )
      Contact( "AutoProcessData".GlobalData.Fixture1CodeOKFlag )
      Contact( "AutoProcessData".GlobalData.Fixture2CodeOKFlag )
      P_Trig( "ChangeOver_DB".P[20] )
      S_Coil( "ChangeOver_DB".Global.AllFixtureScanCompareOk )
      R_Coil( "ChangeOver_DB".Global.ScanFixtureFlag )
   END_RUNG
   RUNG wire#w1
      I_Contact( "AutoProcessData".GlobalData.Table1CodeOKFlag )
      I_Contact( "AutoProcessData".GlobalData.Table2CodeOKFlag )
      I_Contact( "AutoProcessData".GlobalData.Robot1GripperCodeOKFlag )
      I_Contact( "AutoProcessData".GlobalData.Robot2GripperCodeOKFlag )
      I_Contact( "AutoProcessData".GlobalData.Robot3GripperCodeOKFlag )
      I_Contact( "AutoProcessData".GlobalData.Fixture1CodeOKFlag )
      I_Contact( "AutoProcessData".GlobalData.Fixture2CodeOKFlag )
      R_Coil( "ChangeOver_DB".Global.AllFixtureScanCompareOk )
   END_RUNG
   // the same network as SCL:
   #_w1 := "AlwaysTRUE" AND "AutoProcessData".GlobalData.Table1CodeOKFlag AND "AutoProcessData".GlobalData.Table2CodeOKFlag AND "AutoProcessData".GlobalData.Robot1GripperCodeOKFlag AND "AutoProcessData".GlobalData.Robot2GripperCodeOKFlag AND "AutoProcessData".GlobalData.Robot3GripperCodeOKFlag AND "AutoProcessData".GlobalData.Fixture1CodeOKFlag AND "AutoProcessData".GlobalData.Fixture2CodeOKFlag;
   #_w2 := #_w1 AND NOT "ChangeOver_DB".P[20];   // rising edge
   "ChangeOver_DB".P[20] := #_w1;
   IF #_w2 THEN
       "ChangeOver_DB".Global.AllFixtureScanCompareOk := TRUE;
       "ChangeOver_DB".Global.ScanFixtureFlag := FALSE;
   END_IF;
   IF "AlwaysTRUE" AND NOT "AutoProcessData".GlobalData.Table1CodeOKFlag AND NOT "AutoProcessData".GlobalData.Table2CodeOKFlag AND NOT "AutoProcessData".GlobalData.Robot1GripperCodeOKFlag AND NOT "AutoProcessData".GlobalData.Robot2GripperCodeOKFlag AND NOT "AutoProcessData".GlobalData.Robot3GripperCodeOKFlag AND NOT "AutoProcessData".GlobalData.Fixture1CodeOKFlag AND NOT "AutoProcessData".GlobalData.Fixture2CodeOKFlag THEN
       "ChangeOver_DB".Global.AllFixtureScanCompareOk := FALSE;
   END_IF;
END_REGION

REGION Network 24: ---------------------------------- Manual mode Set maintenance pos / Home pos req ------------------------------------------
END_REGION

REGION Network 25: Robot1 Maintenance Pos Req
   RUNG wire#powerrail
      Contact( "AlwaysTRUE" )
      wire#w1
      Contact( "ChangeOver_DB".Robot_1.HMI_MaintenancePosReqSel )
      I_Contact( "KukaRobot1_CtrlDB".sROBtoPLC.User.Cycle.DO297_MaintainInside )
      S_Coil( "ChangeOver_DB".Robot_1.MaintenancePosReqSelFlag )
   END_RUNG
   RUNG wire#w1
      Contact( "ChangeOver_DB".Robot_1.MaintenancePosReqSelFlag )
      wire#w2
      Contact( "KukaRobot2_CtrlDB".sROBtoPLC.User.Cycle.DO298_MaintainFinish )
      wire#w3
      Contact( "ChangeOver_DB".Robot_1.NoTaskRunning )
      Contact( "ChangeOver_DB".Robot_2.NoTaskRunning )
      { S7_Templates := "time_type := Time" } "ChangeOver_DB"."Time"[0].TON(pt := T#500MS, et =>)
      Coil( "ChangeOver_DB".Robot_1.HMI_MaintenancePosActive )
   END_RUNG
   RUNG wire#w2
      Contact( "KukaRobot2_CtrlDB".sROBtoPLC.Sys.SO.IN_HOME )
   END_RUNG wire#w3
   // the same network as SCL:
   IF "AlwaysTRUE" AND "ChangeOver_DB".Robot_1.HMI_MaintenancePosReqSel AND NOT "KukaRobot1_CtrlDB".sROBtoPLC.User.Cycle.DO297_MaintainInside THEN
       "ChangeOver_DB".Robot_1.MaintenancePosReqSelFlag := TRUE;
   END_IF;
   "ChangeOver_DB"."Time"[0].TON(IN := "AlwaysTRUE" AND "ChangeOver_DB".Robot_1.MaintenancePosReqSelFlag AND ("KukaRobot2_CtrlDB".sROBtoPLC.User.Cycle.DO298_MaintainFinish OR "KukaRobot2_CtrlDB".sROBtoPLC.Sys.SO.IN_HOME) AND "ChangeOver_DB".Robot_1.NoTaskRunning AND "ChangeOver_DB".Robot_2.NoTaskRunning,
                           PT := T#500MS);
   "ChangeOver_DB".Robot_1.HMI_MaintenancePosActive := "ChangeOver_DB"."Time"[0].Q;
END_REGION

REGION Network 26: Robot2 Maintenance Pos Req
   RUNG wire#powerrail
      Contact( "AlwaysTRUE" )
      wire#w1
      Contact( "ChangeOver_DB".Robot_2.HMI_MaintenancePosReqSel )
      I_Contact( "KukaRobot2_CtrlDB".sROBtoPLC.User.Cycle.DO297_MaintainInside )
      P_Trig( "AutoProcessControl".P[39] )
      S_Coil( "ChangeOver_DB".Robot_2.MaintenancePosReqSelFlag )
   END_RUNG
   RUNG wire#w1
      Contact( "ChangeOver_DB".Robot_2.MaintenancePosReqSelFlag )
      wire#w2
      Contact( "KukaRobot3_CtrlDB".sROBtoPLC.User.Cycle.DO298_MaintainFinish )
      wire#w3
      Contact( "ChangeOver_DB".Robot_2.NoTaskRunning )
      Contact( "ChangeOver_DB".Robot_3.NoTaskRunning )
      { S7_Templates := "time_type := Time" } "ChangeOver_DB"."Time"[1].TON(pt := T#500MS, et =>)
      Coil( "ChangeOver_DB".Robot_2.HMI_MaintenancePosActive )
   END_RUNG
   RUNG wire#w2
      Contact( "KukaRobot3_CtrlDB".sROBtoPLC.Sys.SO.IN_HOME )
   END_RUNG wire#w3
   // the same network as SCL:
   #_w1 := "AlwaysTRUE" AND "ChangeOver_DB".Robot_2.HMI_MaintenancePosReqSel AND NOT "KukaRobot2_CtrlDB".sROBtoPLC.User.Cycle.DO297_MaintainInside;
   #_w2 := #_w1 AND NOT "AutoProcessControl".P[39];   // rising edge
   "AutoProcessControl".P[39] := #_w1;
   IF #_w2 THEN "ChangeOver_DB".Robot_2.MaintenancePosReqSelFlag := TRUE; END_IF;
   "ChangeOver_DB"."Time"[1].TON(IN := "AlwaysTRUE" AND "ChangeOver_DB".Robot_2.MaintenancePosReqSelFlag AND ("KukaRobot3_CtrlDB".sROBtoPLC.User.Cycle.DO298_MaintainFinish OR "KukaRobot3_CtrlDB".sROBtoPLC.Sys.SO.IN_HOME) AND "ChangeOver_DB".Robot_2.NoTaskRunning AND "ChangeOver_DB".Robot_3.NoTaskRunning,
                           PT := T#500MS);
   "ChangeOver_DB".Robot_2.HMI_MaintenancePosActive := "ChangeOver_DB"."Time"[1].Q;
END_REGION

REGION Network 27: Robot3 Maintenance Pos Req
   RUNG wire#powerrail
      Contact( "AlwaysTRUE" )
      wire#w1
      Contact( "ChangeOver_DB".Robot_3.HMI_MaintenancePosReqSel )
      I_Contact( "KukaRobot3_CtrlDB".sROBtoPLC.User.Cycle.DO297_MaintainInside )
      P_Trig( "AutoProcessControl".P[38] )
      S_Coil( "ChangeOver_DB".Robot_3.MaintenancePosReqSelFlag )
   END_RUNG
   RUNG wire#w1
      Contact( "ChangeOver_DB".Robot_3.MaintenancePosReqSelFlag )
      Contact( "ChangeOver_DB".Robot_3.NoTaskRunning )
      { S7_Templates := "time_type := Time" } "ChangeOver_DB"."Time"[3].TON(pt := T#500MS, et =>)
      Coil( "ChangeOver_DB".Robot_3.HMI_MaintenancePosActive )
   END_RUNG
   // the same network as SCL:
   #_w1 := "AlwaysTRUE" AND "ChangeOver_DB".Robot_3.HMI_MaintenancePosReqSel AND NOT "KukaRobot3_CtrlDB".sROBtoPLC.User.Cycle.DO297_MaintainInside;
   #_w2 := #_w1 AND NOT "AutoProcessControl".P[38];   // rising edge
   "AutoProcessControl".P[38] := #_w1;
   IF #_w2 THEN "ChangeOver_DB".Robot_3.MaintenancePosReqSelFlag := TRUE; END_IF;
   "ChangeOver_DB"."Time"[3].TON(IN := "AlwaysTRUE" AND "ChangeOver_DB".Robot_3.MaintenancePosReqSelFlag AND "ChangeOver_DB".Robot_3.NoTaskRunning,
                           PT := T#500MS);
   "ChangeOver_DB".Robot_3.HMI_MaintenancePosActive := "ChangeOver_DB"."Time"[3].Q;
END_REGION

REGION Network 28: Station empty
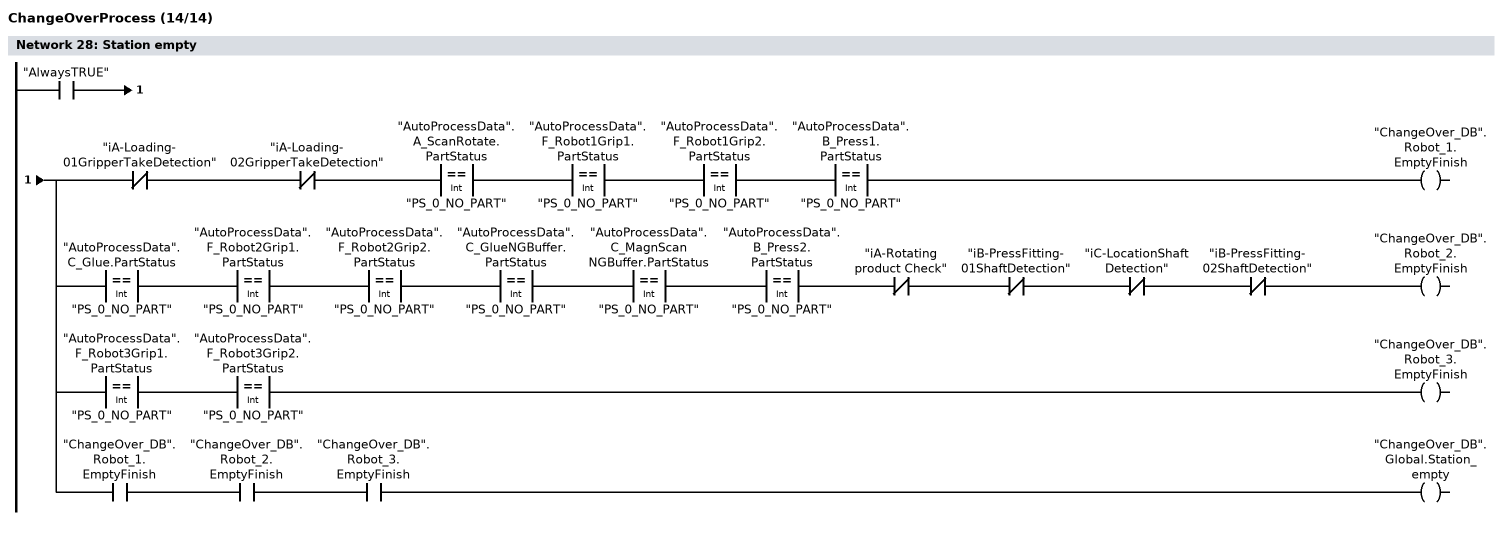
   RUNG wire#powerrail
      Contact( "AlwaysTRUE" )
      wire#w1
      I_Contact( "iA-Loading-01GripperTakeDetection" )
      I_Contact( "iA-Loading-02GripperTakeDetection" )
      { S7_Templates := "SrcType := Int" } EQ_Contact(in1 := "AutoProcessData".A_ScanRotate.PartStatus, in2 := "PS_0_NO_PART")
      { S7_Templates := "SrcType := Int" } EQ_Contact(in1 := "AutoProcessData".F_Robot1Grip1.PartStatus, in2 := "PS_0_NO_PART")
      { S7_Templates := "SrcType := Int" } EQ_Contact(in1 := "AutoProcessData".F_Robot1Grip2.PartStatus, in2 := "PS_0_NO_PART")
      { S7_Templates := "SrcType := Int" } EQ_Contact(in1 := "AutoProcessData".B_Press1.PartStatus, in2 := "PS_0_NO_PART")
      Coil( "ChangeOver_DB".Robot_1.EmptyFinish )
   END_RUNG
   RUNG wire#w1
      { S7_Templates := "SrcType := Int" } EQ_Contact(in1 := "AutoProcessData".C_Glue.PartStatus, in2 := "PS_0_NO_PART")
      { S7_Templates := "SrcType := Int" } EQ_Contact(in1 := "AutoProcessData".F_Robot2Grip1.PartStatus, in2 := "PS_0_NO_PART")
      { S7_Templates := "SrcType := Int" } EQ_Contact(in1 := "AutoProcessData".F_Robot2Grip2.PartStatus, in2 := "PS_0_NO_PART")
      { S7_Templates := "SrcType := Int" } EQ_Contact(in1 := "AutoProcessData".C_GlueNGBuffer.PartStatus, in2 := "PS_0_NO_PART")
      { S7_Templates := "SrcType := Int" } EQ_Contact(in1 := "AutoProcessData".C_MagnScanNGBuffer.PartStatus, in2 := "PS_0_NO_PART")
      { S7_Templates := "SrcType := Int" } EQ_Contact(in1 := "AutoProcessData".B_Press2.PartStatus, in2 := "PS_0_NO_PART")
      I_Contact( "iA-Rotating product Check" )
      I_Contact( "iB-PressFitting-01ShaftDetection" )
      I_Contact( "iC-LocationShaftDetection" )
      I_Contact( "iB-PressFitting-02ShaftDetection" )
      Coil( "ChangeOver_DB".Robot_2.EmptyFinish )
   END_RUNG
   RUNG wire#w1
      { S7_Templates := "SrcType := Int" } EQ_Contact(in1 := "AutoProcessData".F_Robot3Grip1.PartStatus, in2 := "PS_0_NO_PART")
      { S7_Templates := "SrcType := Int" } EQ_Contact(in1 := "AutoProcessData".F_Robot3Grip2.PartStatus, in2 := "PS_0_NO_PART")
      Coil( "ChangeOver_DB".Robot_3.EmptyFinish )
   END_RUNG
   RUNG wire#w1
      Contact( "ChangeOver_DB".Robot_1.EmptyFinish )
      Contact( "ChangeOver_DB".Robot_2.EmptyFinish )
      Contact( "ChangeOver_DB".Robot_3.EmptyFinish )
      Coil( "ChangeOver_DB".Global.Station_empty )
   END_RUNG
   // the same network as SCL:
   "ChangeOver_DB".Robot_1.EmptyFinish := "AlwaysTRUE" AND NOT "iA-Loading-01GripperTakeDetection" AND NOT "iA-Loading-02GripperTakeDetection" AND ("AutoProcessData".A_ScanRotate.PartStatus = "PS_0_NO_PART") AND ("AutoProcessData".F_Robot1Grip1.PartStatus = "PS_0_NO_PART") AND ("AutoProcessData".F_Robot1Grip2.PartStatus = "PS_0_NO_PART") AND ("AutoProcessData".B_Press1.PartStatus = "PS_0_NO_PART");
   "ChangeOver_DB".Robot_2.EmptyFinish := "AlwaysTRUE" AND ("AutoProcessData".C_Glue.PartStatus = "PS_0_NO_PART") AND ("AutoProcessData".F_Robot2Grip1.PartStatus = "PS_0_NO_PART") AND ("AutoProcessData".F_Robot2Grip2.PartStatus = "PS_0_NO_PART") AND ("AutoProcessData".C_GlueNGBuffer.PartStatus = "PS_0_NO_PART") AND ("AutoProcessData".C_MagnScanNGBuffer.PartStatus = "PS_0_NO_PART") AND ("AutoProcessData".B_Press2.PartStatus = "PS_0_NO_PART") AND NOT "iA-Rotating product Check" AND NOT "iB-PressFitting-01ShaftDetection" AND NOT "iC-LocationShaftDetection" AND NOT "iB-PressFitting-02ShaftDetection";
   "ChangeOver_DB".Robot_3.EmptyFinish := "AlwaysTRUE" AND ("AutoProcessData".F_Robot3Grip1.PartStatus = "PS_0_NO_PART") AND ("AutoProcessData".F_Robot3Grip2.PartStatus = "PS_0_NO_PART");
   "ChangeOver_DB".Global.Station_empty := "AlwaysTRUE" AND "ChangeOver_DB".Robot_1.EmptyFinish AND "ChangeOver_DB".Robot_2.EmptyFinish AND "ChangeOver_DB".Robot_3.EmptyFinish;
END_REGION
END_FUNCTION

FUNCTION_BLOCK "ST10_Flow1_A1TableScan"   // FB1071, GRAPH
// stored: AcknowledgeErrorsRequired false, AutoNumber false, GraphVersion 6.0, InitialValuesAcquisition false, SetENOAutomatically false
   // inherited from GRAPH_BASE
   VAR_INPUT
      iSysInface : "RCS_SysComInterface_V1";
   END_VAR
   VAR_IN_OUT
      ioPM_Inface : "RCS_PMInterface_V1";
      ioStatus : Int;
   END_VAR
   VAR
      sCtrlMode { S7_SetPoint := 'True'} : "SysFlowCtrlGraph";
      sUpdMES_Data : Bool;   // 更新MES数据
      工件放行中 : Bool;
      前站站号 { ExternalAccessible := 'False'; ExternalVisible := 'False'; ExternalWritable := 'False'} : UInt;
      本站站号 { ExternalAccessible := 'False'; ExternalVisible := 'False'; ExternalWritable := 'False'} : UInt;
      弹窗Temp : Array[1..10] of Int;
      AlarmID : Int;
      TON { S7_SetPoint := 'True'} : Array[0..10] of TON_TIME;
      TOF { S7_SetPoint := 'True'} : Array[0..10] of TOF_TIME;
      sUP { S7_SetPoint := 'True'} : Array[0..10] of Bool;
      更新RFID完成 : Bool;
   END_VAR
   VAR_TEMP
      Tempresult : USInt;
      本站站号乘10 : UInt;
   END_VAR
   // // TON[0] : 托盘流入1托盘到位传感器 / iA-Rotating product Check
   // // TON[1] : 托盘流入1托盘到位传感器
   // // TON[2] : 托盘流入1产品有无传感器
   // // TON[3] : 托盘流入1产品有无传感器
   // // TON[4] : 托盘流入1姿态检测光电2
   // // TON[5] : 托盘流入1姿态检测光电3
   // // TON[0].Q : 托盘流入1托盘到位 / iA-Rotating product Check
   // // TON[1].Q : 托盘流入1托盘无
   // // TON[2].Q : 托盘流入1有产品
   // // TON[3].Q : 托盘流入1无产品
   // // TON[4].Q : 托盘流入1姿态检测光电2
   // // TON[5].Q : 托盘流入1姿态检测光电3
   // // TOF[1] : iA-Rotating product Check
BEGIN
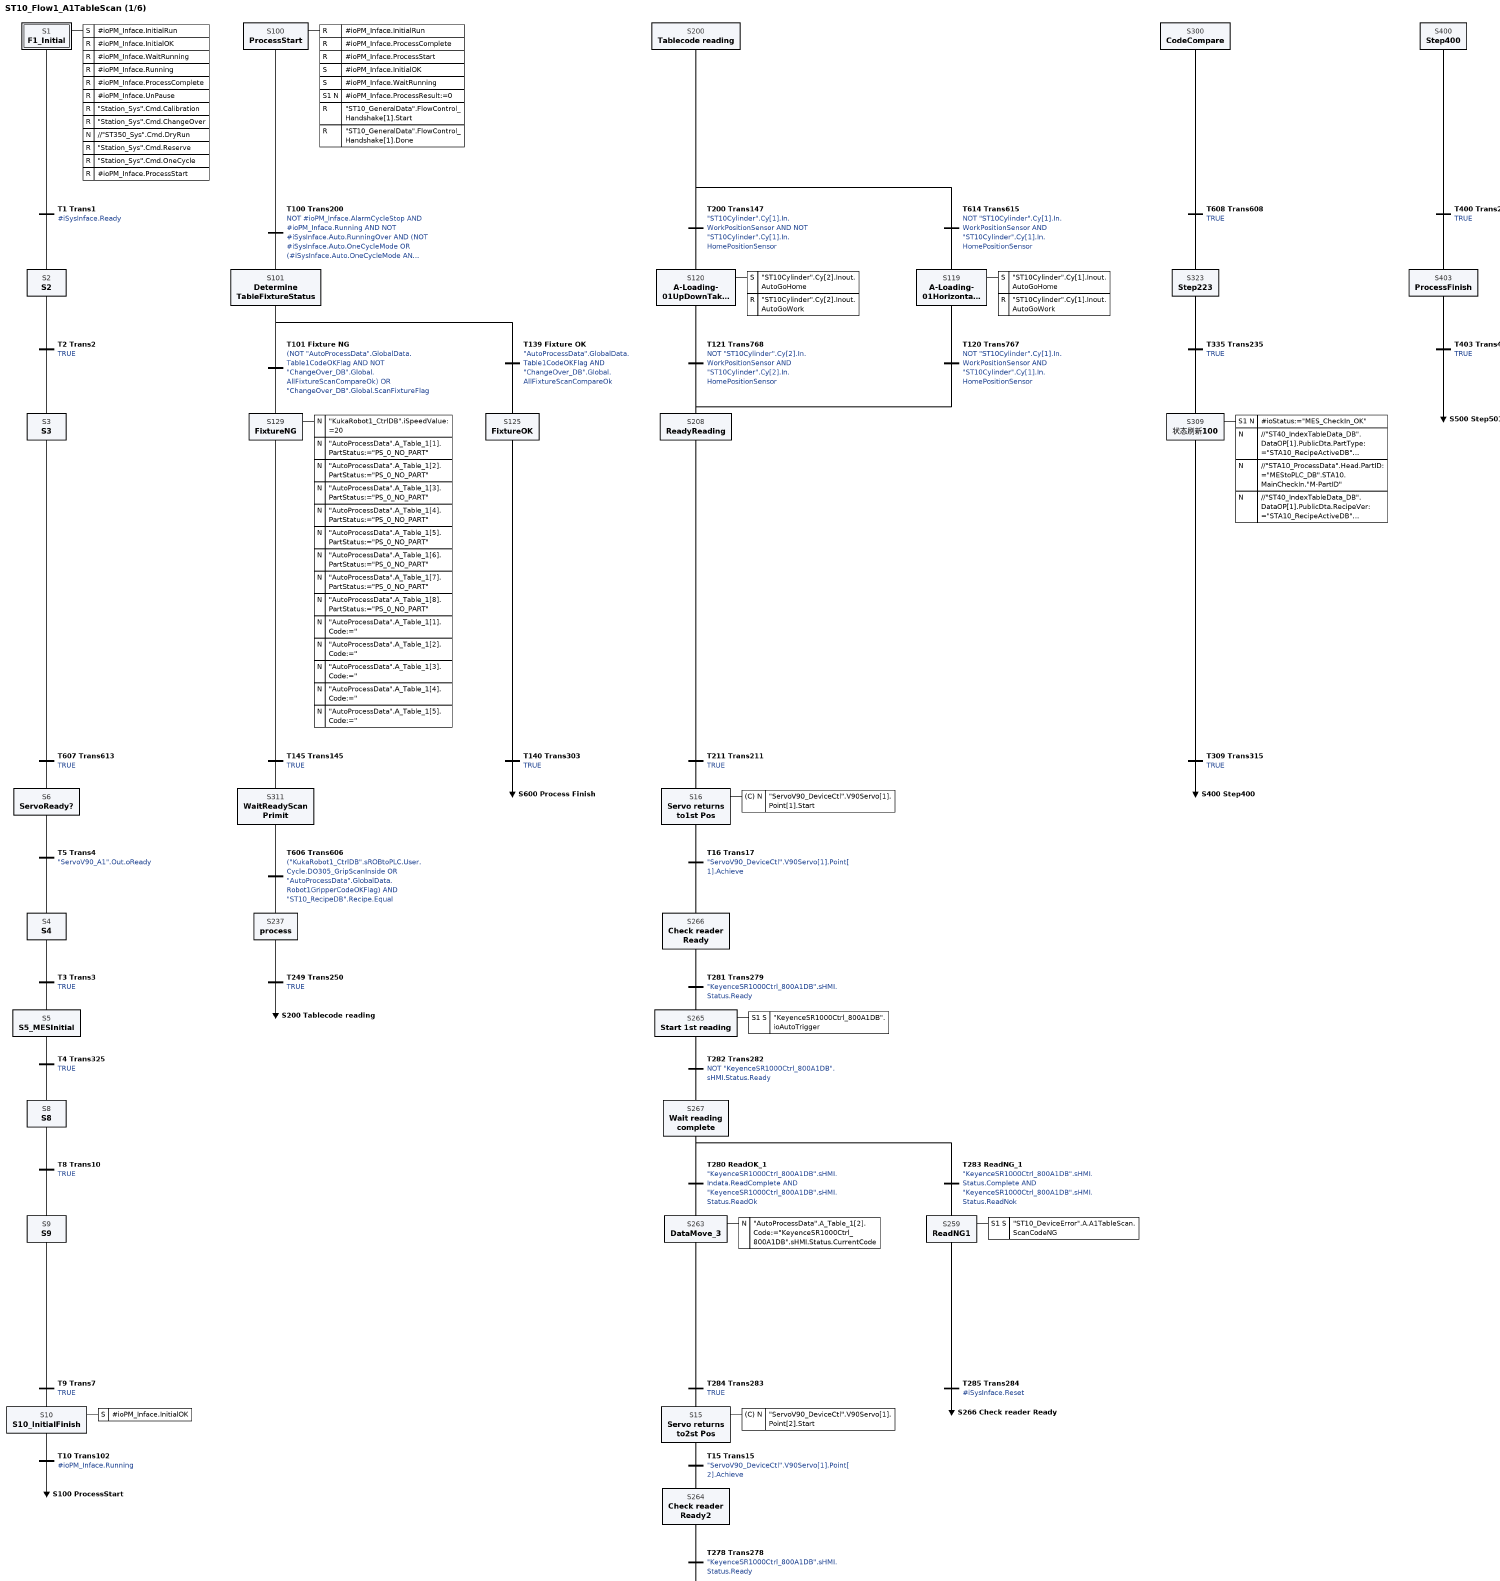
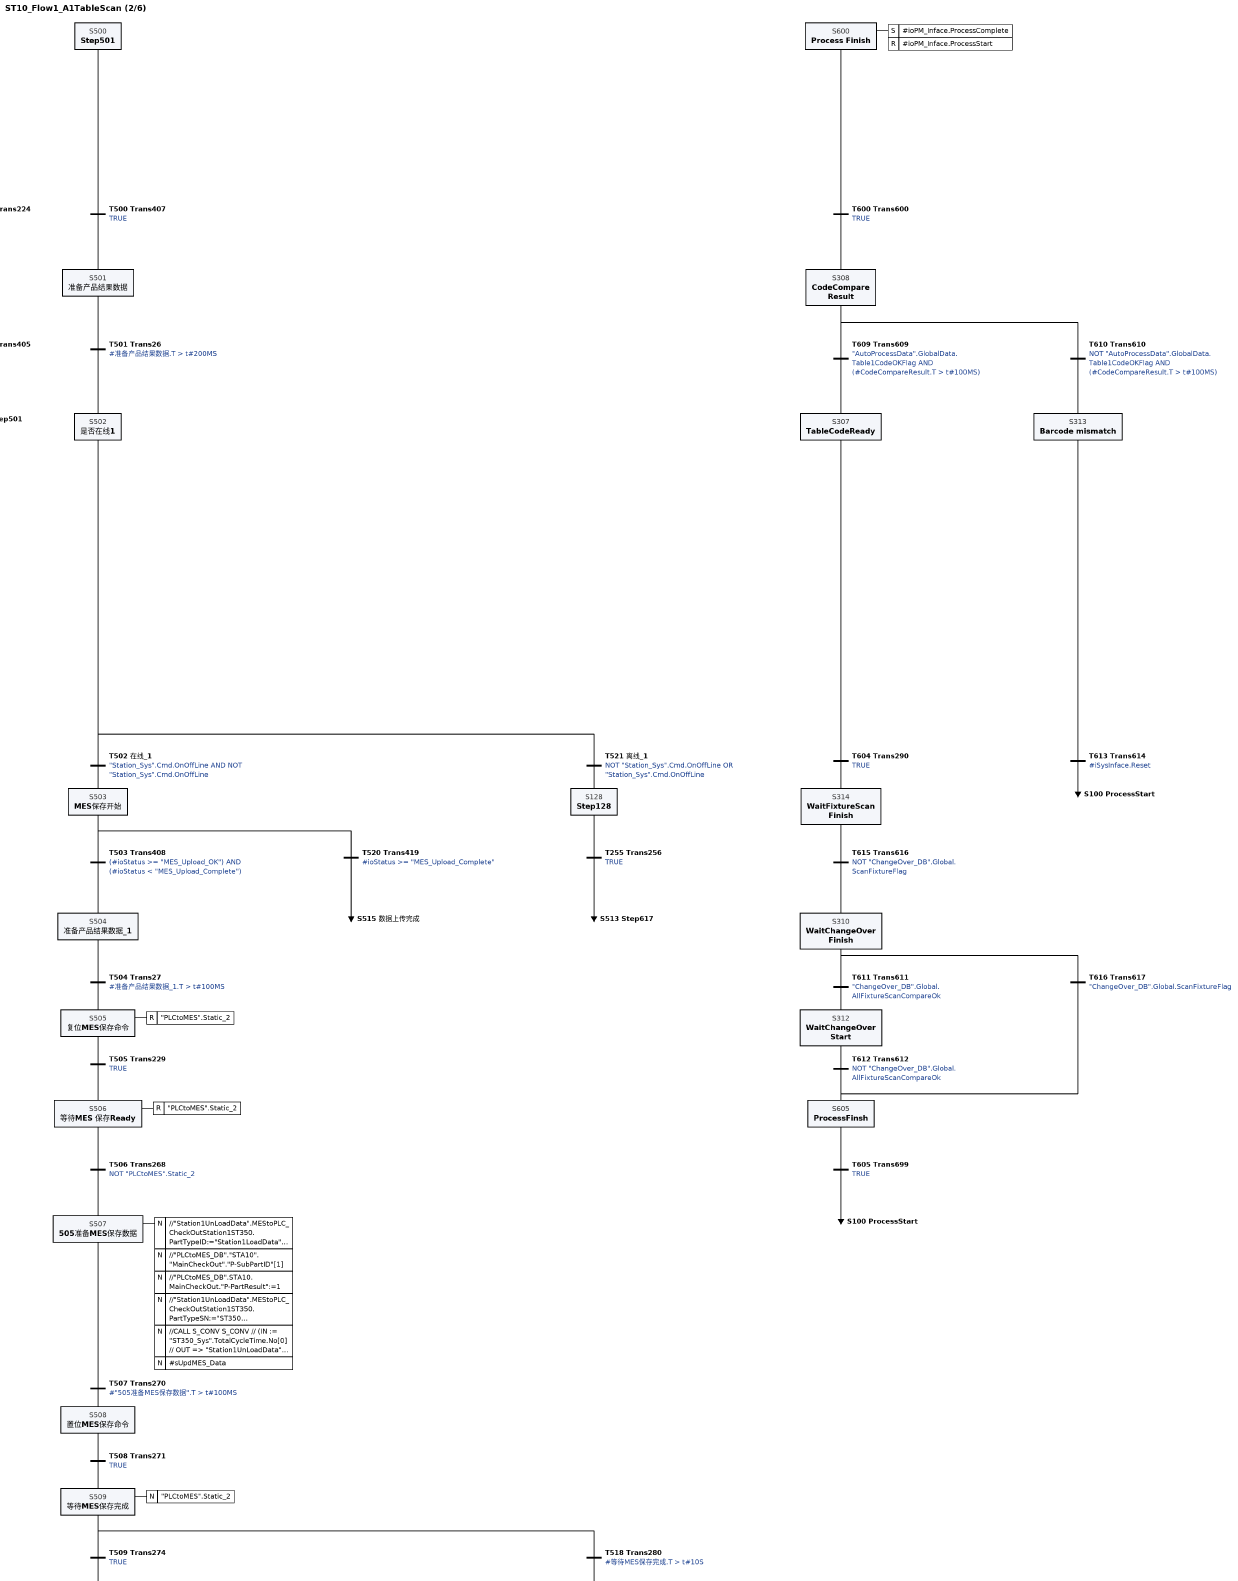
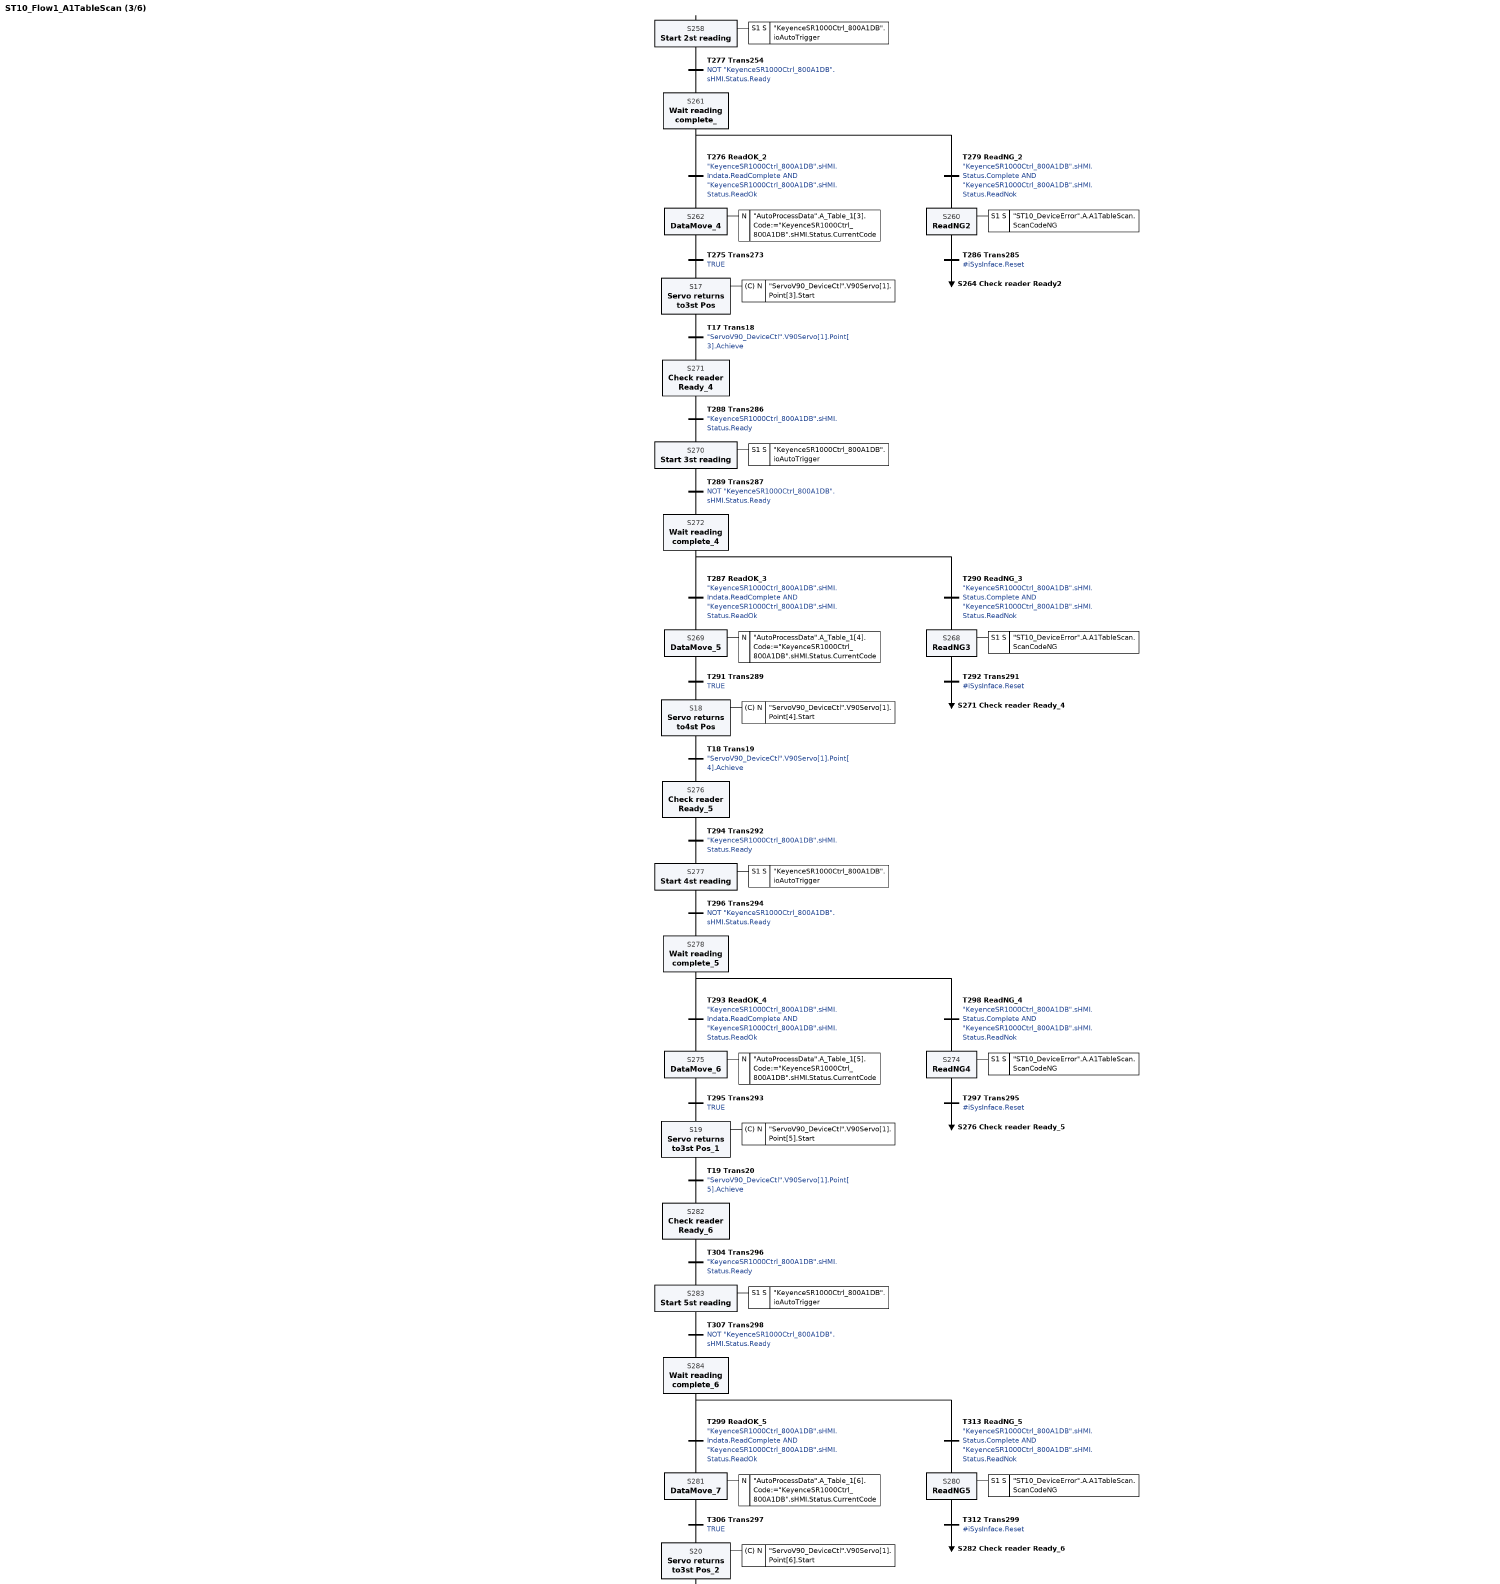
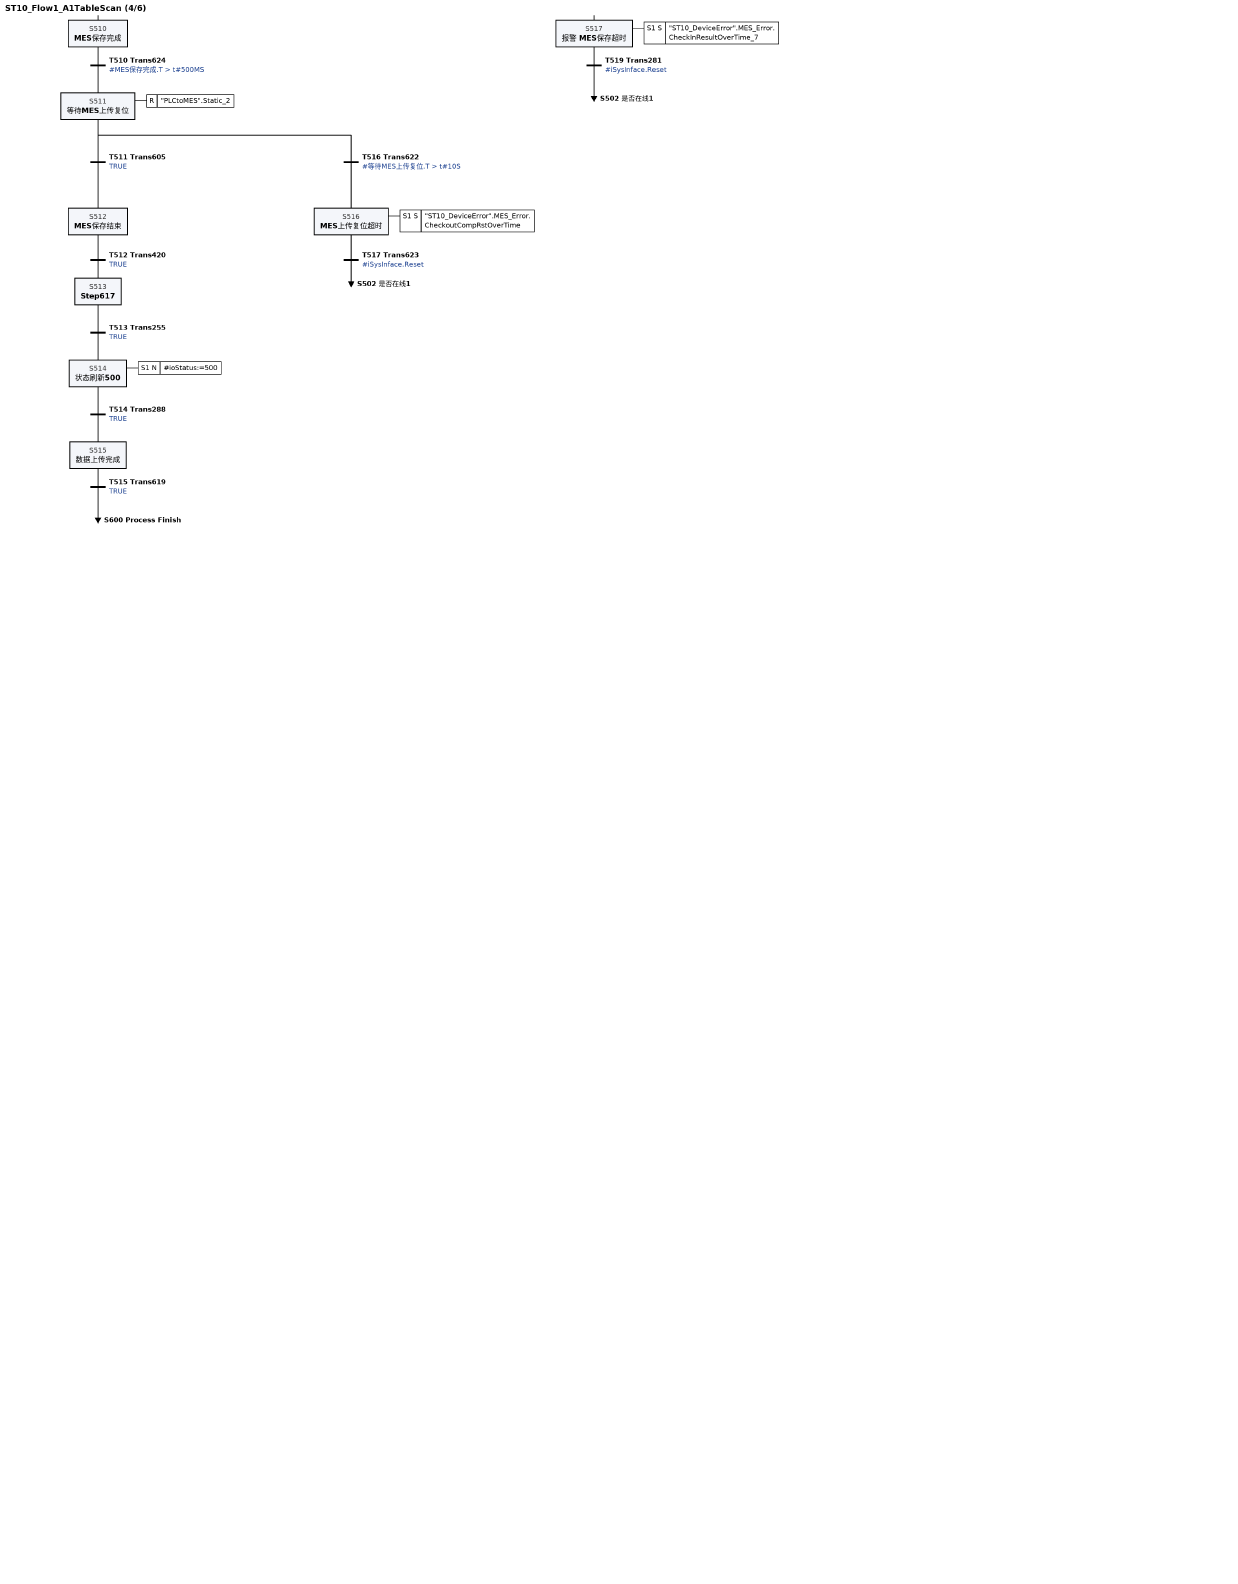
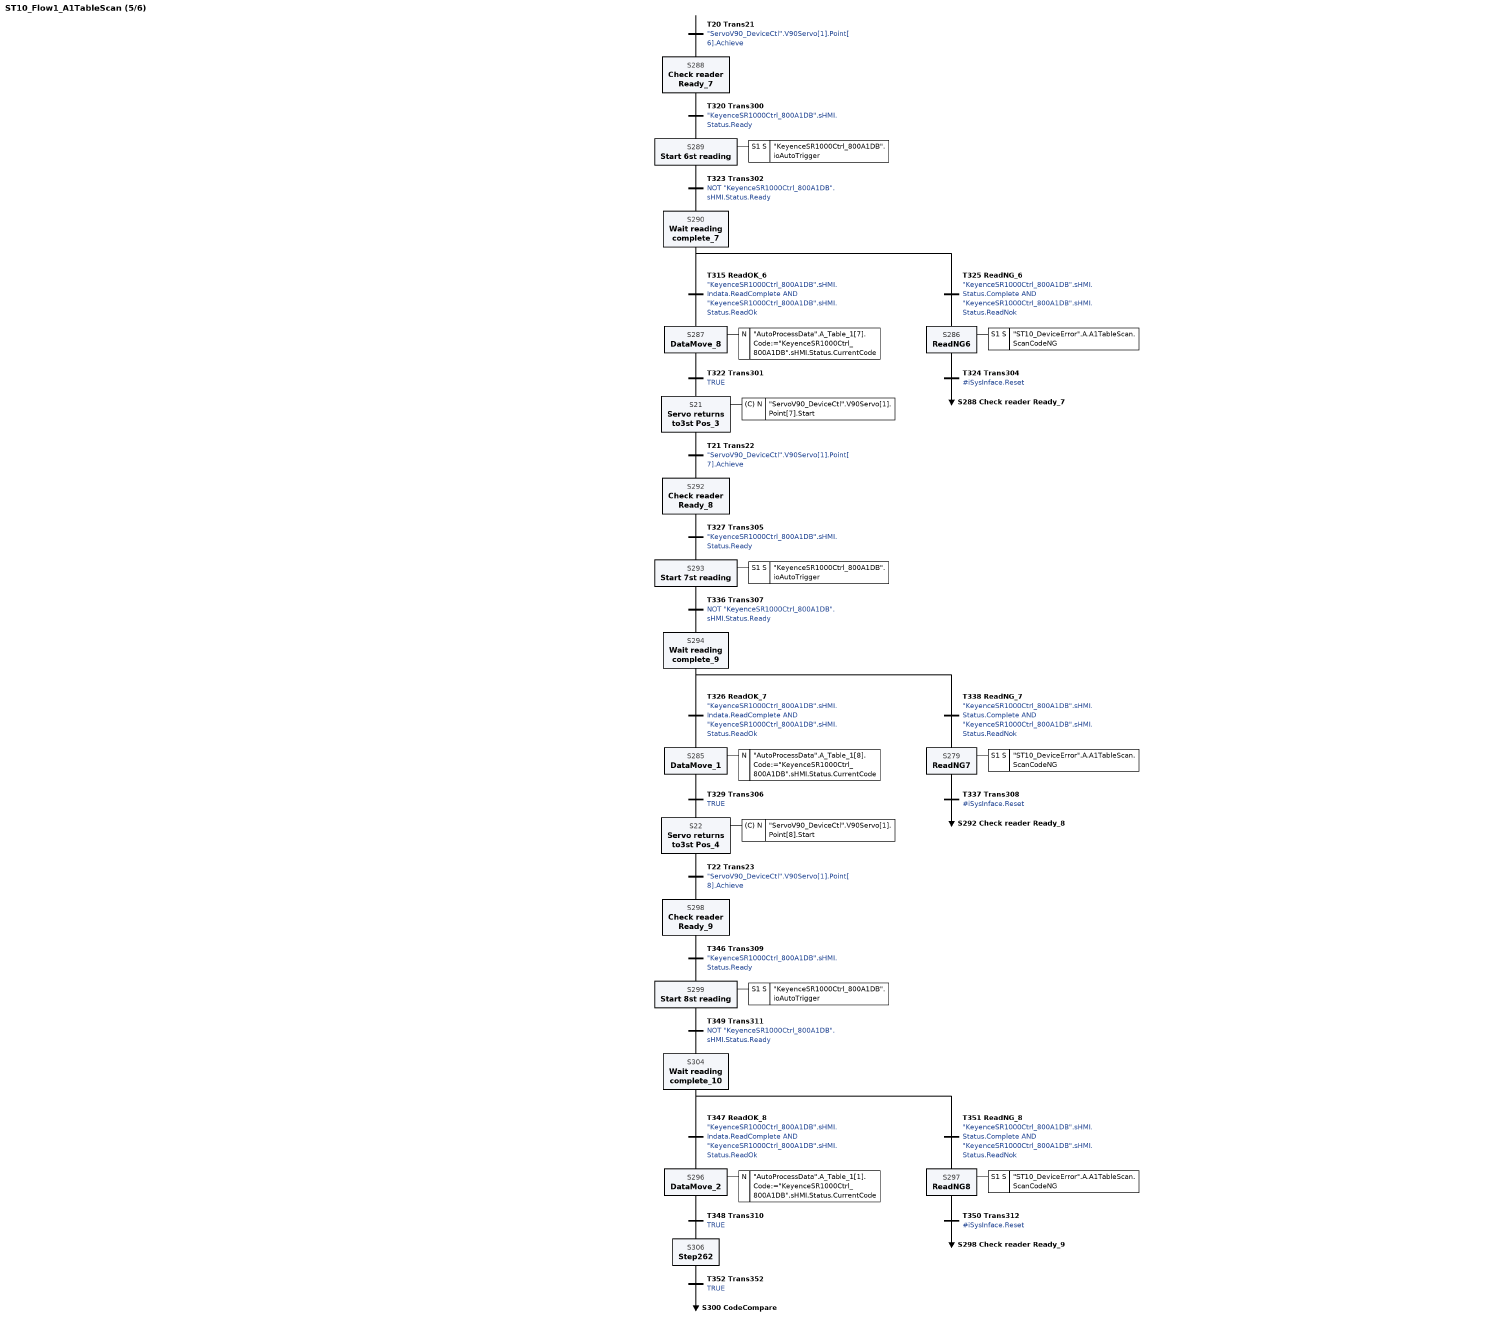
   // permanent pre-instructions
   NETWORK 1
      #TON[10].TON(IN := "AlwaysTRUE" AND "Station_Sys".Alarm.ImmediatelyStop, PT := T#300ms);
      #ioPM_Inface.AlarmImdilyStop := #TON[10].Q;
      #ioPM_Inface.AlarmCycleStop := "AlwaysTRUE" AND "Station_Sys".Alarm.CycleStop;
   NETWORK 2
      IF NOT False THEN
          #sCtrlMode(iSysInface := #iSysInface, ioPM_Inface := #ioPM_Inface, ioGraphCtrl := #RT_DATA.MOP);   // "SysFlowCtrlGraph"
      END_IF;
   NETWORK 3
      #TON[0].TON(IN := "AlwaysTRUE" AND "iA-Rotating product Check", PT := t#500ms);   // 工位11有托盘
      #TON[1].TOF(IN := "AlwaysTRUE" AND NOT "iA-Rotating product Check", PT := T#300ms);   // 工位无托盘
      #TON[2].TON(IN := "AlwaysTRUE", PT := T#300ms);
      #TON[3].TON(IN := "AlwaysTRUE", PT := T#300ms);
      #TON[4].TON(IN := "AlwaysTRUE", PT := T#300ms);
      #TON[5].TON(IN := "AlwaysTRUE", PT := T#300ms);
   NETWORK 4
      #前站站号 := 345;
      #本站站号 := 350;

   // sequencer 1: S01-S99 初始化 / S01-S99 Initial
   INITIAL_STEP F1_Initial:   // S1, max time T#10S, warning time T#7S
              S    #ioPM_Inface.InitialRun
              R    #ioPM_Inface.InitialOK
              R    #ioPM_Inface.WaitRunning
              R    #ioPM_Inface.Running
              R    #ioPM_Inface.ProcessComplete
              R    #ioPM_Inface.UnPause
              R    "Station_Sys".Cmd.Calibration
              R    "Station_Sys".Cmd.ChangeOver
                   //"ST350_Sys".Cmd.DryRun
              R    "Station_Sys".Cmd.Reserve
              R    "Station_Sys".Cmd.OneCycle
              R    #ioPM_Inface.ProcessStart
   END_STEP
   TRANSITION Trans1 FROM F1_Initial TO S2   // T1
      := #iSysInface.Ready;
   END_TRANSITION
   STEP S2:   // S2, max time T#10S, warning time T#7S
   END_STEP
   TRANSITION Trans2 FROM S2 TO S3   // T2
      := TRUE;
   END_TRANSITION
   STEP S4:   // S4, max time T#10S, warning time T#7S
   END_STEP
   TRANSITION Trans3 FROM S4 TO S5_MESInitial   // T3
      := TRUE;
   END_TRANSITION
   STEP S5_MESInitial:   // S5, max time T#10S, warning time T#7S
   END_STEP
   TRANSITION Trans325 FROM S5_MESInitial TO S8   // T4
      := TRUE;
   END_TRANSITION
   STEP S10_InitialFinish:   // S10, max time T#10S, warning time T#7S
              S    #ioPM_Inface.InitialOK
   END_STEP
   TRANSITION Trans102 FROM S10_InitialFinish TO ProcessStart   // T10, jump
      := #ioPM_Inface.Running;
   END_TRANSITION
   STEP S3:   // S3, max time T#10S, warning time T#7S
   END_STEP
   TRANSITION Trans613 FROM S3 TO "ServoReady?"   // T607
      := TRUE;
   END_TRANSITION
   STEP S8:   // S8, max time T#10S, warning time T#7S
   END_STEP
   TRANSITION Trans10 FROM S8 TO S9   // T8
      := TRUE;
   END_TRANSITION
   STEP S9:   // S9, max time T#10S, warning time T#7S
   END_STEP
   TRANSITION Trans7 FROM S9 TO S10_InitialFinish   // T9
      := TRUE;
   END_TRANSITION
   STEP "ServoReady?":   // S6, max time T#10S, warning time T#7S
   END_STEP
   TRANSITION Trans4 FROM "ServoReady?" TO S4   // T5
      := "ServoV90_A1".Out.oReady;
   END_TRANSITION

   // sequencer 2: S100-S199 等待到位 / S100-S199 CheckPartStatus
   STEP ProcessStart:   // S100, max time T#10S, warning time T#7S
      // 自动等待开始运行
              R    #ioPM_Inface.InitialRun
              R    #ioPM_Inface.ProcessComplete
              R    #ioPM_Inface.ProcessStart
              S    #ioPM_Inface.InitialOK
              S    #ioPM_Inface.WaitRunning
          S1  N    #ioPM_Inface.ProcessResult:=0
              R    "ST10_GeneralData".FlowControl_Handshake[1].Start
              R    "ST10_GeneralData".FlowControl_Handshake[1].Done
   END_STEP
   TRANSITION Trans200 FROM ProcessStart TO "Determine TableFixtureStatus"   // T100
      := NOT #ioPM_Inface.AlarmCycleStop AND #ioPM_Inface.Running AND NOT #iSysInface.Auto.RunningOver AND (NOT #iSysInface.Auto.OneCycleMode OR (#iSysInface.Auto.OneCycleMode AND #ioPM_Inface.TriggerOneCycle));
   END_TRANSITION
   STEP process:   // S237, max time T#10S, warning time T#7S
   END_STEP
   TRANSITION Trans250 FROM process TO "Tablecode reading"   // T249, jump
      := TRUE;
   END_TRANSITION
   STEP "Determine TableFixtureStatus":   // S101, max time T#10S, warning time T#7S
   END_STEP
   TRANSITION "Fixture NG" FROM "Determine TableFixtureStatus" TO FixtureNG   // T101
      := (NOT "AutoProcessData".GlobalData.Table1CodeOKFlag AND NOT "ChangeOver_DB".Global.AllFixtureScanCompareOk) OR "ChangeOver_DB".Global.ScanFixtureFlag;
   END_TRANSITION
   TRANSITION "Fixture OK" FROM "Determine TableFixtureStatus" TO FixtureOK   // T139
      := "AutoProcessData".GlobalData.Table1CodeOKFlag AND "ChangeOver_DB".Global.AllFixtureScanCompareOk;
   END_TRANSITION
   STEP FixtureOK:   // S125, max time T#10S, warning time T#7S
   END_STEP
   TRANSITION Trans303 FROM FixtureOK TO "Process Finish"   // T140, jump
      := TRUE;
   END_TRANSITION
   STEP FixtureNG:   // S129, max time T#10S, warning time T#7S
              N    "KukaRobot1_CtrlDB".iSpeedValue:=20
              N    "AutoProcessData".A_Table_1[1].PartStatus:="PS_0_NO_PART"
              N    "AutoProcessData".A_Table_1[2].PartStatus:="PS_0_NO_PART"
              N    "AutoProcessData".A_Table_1[3].PartStatus:="PS_0_NO_PART"
              N    "AutoProcessData".A_Table_1[4].PartStatus:="PS_0_NO_PART"
              N    "AutoProcessData".A_Table_1[5].PartStatus:="PS_0_NO_PART"
              N    "AutoProcessData".A_Table_1[6].PartStatus:="PS_0_NO_PART"
              N    "AutoProcessData".A_Table_1[7].PartStatus:="PS_0_NO_PART"
              N    "AutoProcessData".A_Table_1[8].PartStatus:="PS_0_NO_PART"
              N    "AutoProcessData".A_Table_1[1].Code:=''
              N    "AutoProcessData".A_Table_1[2].Code:=''
              N    "AutoProcessData".A_Table_1[3].Code:=''
              N    "AutoProcessData".A_Table_1[4].Code:=''
              N    "AutoProcessData".A_Table_1[5].Code:=''
              N    "AutoProcessData".A_Table_1[6].Code:=''
              N    "AutoProcessData".A_Table_1[7].Code:=''
              N    "AutoProcessData".A_Table_1[8].Code:=''
   END_STEP
   TRANSITION Trans145 FROM FixtureNG TO WaitReadyScanPrimit   // T145
      := TRUE;
   END_TRANSITION
   STEP WaitReadyScanPrimit:   // S311, max time T#10S, warning time T#7S
   END_STEP
   TRANSITION Trans606 FROM WaitReadyScanPrimit TO process   // T606
      := ("KukaRobot1_CtrlDB".sROBtoPLC.User.Cycle.DO305_GripScanInside OR "AutoProcessData".GlobalData.Robot1GripperCodeOKFlag) AND "ST10_RecipeDB".Recipe.Equal;
   END_TRANSITION

   // sequencer 3: S200-S299Tablecode reading
   STEP "Tablecode reading":   // S200, max time T#10S, warning time T#7S
   END_STEP
   TRANSITION Trans147 FROM "Tablecode reading" TO "A-Loading-01UpDownTakeCylinderToHP"   // T200
      := "ST10Cylinder".Cy[1].In.WorkPositionSensor AND NOT "ST10Cylinder".Cy[1].In.HomePositionSensor;
   END_TRANSITION
   TRANSITION Trans615 FROM "Tablecode reading" TO "A-Loading-01HorizontalCylinderToHP"   // T614
      := NOT "ST10Cylinder".Cy[1].In.WorkPositionSensor AND "ST10Cylinder".Cy[1].In.HomePositionSensor;
   END_TRANSITION
   STEP "Start 2st reading":   // S258, max time T#10S, warning time T#7S
          S1  S    "KeyenceSR1000Ctrl_800A1DB".ioAutoTrigger
   END_STEP
   TRANSITION Trans254 FROM "Start 2st reading" TO "Wait reading complete_"   // T277
      := NOT "KeyenceSR1000Ctrl_800A1DB".sHMI.Status.Ready;
   END_TRANSITION
   STEP ReadNG1:   // S259, max time T#10S, warning time T#7S
          S1  S    "ST10_DeviceError".A.A1TableScan.ScanCodeNG
   END_STEP
   TRANSITION Trans284 FROM ReadNG1 TO "Check reader Ready"   // T285, jump
      := #iSysInface.Reset;
   END_TRANSITION
   STEP ReadNG2:   // S260, max time T#10S, warning time T#7S
          S1  S    "ST10_DeviceError".A.A1TableScan.ScanCodeNG
   END_STEP
   TRANSITION Trans285 FROM ReadNG2 TO "Check reader Ready2"   // T286, jump
      := #iSysInface.Reset;
   END_TRANSITION
   STEP DataMove_4:   // S262, max time T#10S, warning time T#7S
              N    "AutoProcessData".A_Table_1[3].Code:="KeyenceSR1000Ctrl_800A1DB".sHMI.Status.CurrentCode
   END_STEP
   TRANSITION Trans273 FROM DataMove_4 TO "Servo returns to3st Pos"   // T275
      := TRUE;
   END_TRANSITION
   STEP "Wait reading complete_":   // S261, max time T#10S, warning time T#7S
   END_STEP
   TRANSITION ReadOK_2 FROM "Wait reading complete_" TO DataMove_4   // T276
      := "KeyenceSR1000Ctrl_800A1DB".sHMI.Indata.ReadComplete AND "KeyenceSR1000Ctrl_800A1DB".sHMI.Status.ReadOk;
   END_TRANSITION
   TRANSITION ReadNG_2 FROM "Wait reading complete_" TO ReadNG2   // T279
      := "KeyenceSR1000Ctrl_800A1DB".sHMI.Status.Complete AND "KeyenceSR1000Ctrl_800A1DB".sHMI.Status.ReadNok;
   END_TRANSITION
   STEP "Servo returns to2st Pos":   // S15, max time T#10S, warning time T#7S
      interlock C := "ServoV90_A1".Out.oReady;
      (C)     N    "ServoV90_DeviceCtl".V90Servo[1].Point[2].Start
   END_STEP
   TRANSITION Trans15 FROM "Servo returns to2st Pos" TO "Check reader Ready2"   // T15
      := "ServoV90_DeviceCtl".V90Servo[1].Point[2].Achieve;
   END_TRANSITION
   STEP ReadyReading:   // S208, max time T#10S, warning time T#7S
   END_STEP
   TRANSITION Trans211 FROM ReadyReading TO "Servo returns to1st Pos"   // T211
      := TRUE;
   END_TRANSITION
   STEP DataMove_3:   // S263, max time T#10S, warning time T#7S
              N    "AutoProcessData".A_Table_1[2].Code:="KeyenceSR1000Ctrl_800A1DB".sHMI.Status.CurrentCode
   END_STEP
   TRANSITION Trans283 FROM DataMove_3 TO "Servo returns to2st Pos"   // T284
      := TRUE;
   END_TRANSITION
   STEP "Servo returns to1st Pos":   // S16, max time T#10S, warning time T#7S
      interlock C := "ServoV90_A1".Out.oReady;
      (C)     N    "ServoV90_DeviceCtl".V90Servo[1].Point[1].Start
   END_STEP
   TRANSITION Trans17 FROM "Servo returns to1st Pos" TO "Check reader Ready"   // T16
      := "ServoV90_DeviceCtl".V90Servo[1].Point[1].Achieve;
   END_TRANSITION
   STEP "Check reader Ready2":   // S264, max time T#10S, warning time T#7S
   END_STEP
   TRANSITION Trans278 FROM "Check reader Ready2" TO "Start 2st reading"   // T278
      := "KeyenceSR1000Ctrl_800A1DB".sHMI.Status.Ready;
   END_TRANSITION
   STEP "Start 1st reading":   // S265, max time T#10S, warning time T#7S
          S1  S    "KeyenceSR1000Ctrl_800A1DB".ioAutoTrigger
   END_STEP
   TRANSITION Trans282 FROM "Start 1st reading" TO "Wait reading complete"   // T282
      := NOT "KeyenceSR1000Ctrl_800A1DB".sHMI.Status.Ready;
   END_TRANSITION
   STEP "Check reader Ready":   // S266, max time T#10S, warning time T#7S
   END_STEP
   TRANSITION Trans279 FROM "Check reader Ready" TO "Start 1st reading"   // T281
      := "KeyenceSR1000Ctrl_800A1DB".sHMI.Status.Ready;
   END_TRANSITION
   STEP ReadNG3:   // S268, max time T#10S, warning time T#7S
          S1  S    "ST10_DeviceError".A.A1TableScan.ScanCodeNG
   END_STEP
   TRANSITION Trans291 FROM ReadNG3 TO "Check reader Ready_4"   // T292, jump
      := #iSysInface.Reset;
   END_TRANSITION
   STEP "Wait reading complete":   // S267, max time T#10S, warning time T#7S
   END_STEP
   TRANSITION ReadOK_1 FROM "Wait reading complete" TO DataMove_3   // T280
      := "KeyenceSR1000Ctrl_800A1DB".sHMI.Indata.ReadComplete AND "KeyenceSR1000Ctrl_800A1DB".sHMI.Status.ReadOk;
   END_TRANSITION
   TRANSITION ReadNG_1 FROM "Wait reading complete" TO ReadNG1   // T283
      := "KeyenceSR1000Ctrl_800A1DB".sHMI.Status.Complete AND "KeyenceSR1000Ctrl_800A1DB".sHMI.Status.ReadNok;
   END_TRANSITION
   STEP DataMove_5:   // S269, max time T#10S, warning time T#7S
              N    "AutoProcessData".A_Table_1[4].Code:="KeyenceSR1000Ctrl_800A1DB".sHMI.Status.CurrentCode
   END_STEP
   TRANSITION Trans289 FROM DataMove_5 TO "Servo returns to4st Pos"   // T291
      := TRUE;
   END_TRANSITION
   STEP "Servo returns to3st Pos":   // S17, max time T#10S, warning time T#7S
      interlock C := "ServoV90_A1".Out.oReady;
      (C)     N    "ServoV90_DeviceCtl".V90Servo[1].Point[3].Start
   END_STEP
   TRANSITION Trans18 FROM "Servo returns to3st Pos" TO "Check reader Ready_4"   // T17
      := "ServoV90_DeviceCtl".V90Servo[1].Point[3].Achieve;
   END_TRANSITION
   STEP "Check reader Ready_4":   // S271, max time T#10S, warning time T#7S
   END_STEP
   TRANSITION Trans286 FROM "Check reader Ready_4" TO "Start 3st reading"   // T288
      := "KeyenceSR1000Ctrl_800A1DB".sHMI.Status.Ready;
   END_TRANSITION
   STEP "Start 3st reading":   // S270, max time T#10S, warning time T#7S
          S1  S    "KeyenceSR1000Ctrl_800A1DB".ioAutoTrigger
   END_STEP
   TRANSITION Trans287 FROM "Start 3st reading" TO "Wait reading complete_4"   // T289
      := NOT "KeyenceSR1000Ctrl_800A1DB".sHMI.Status.Ready;
   END_TRANSITION
   STEP "Wait reading complete_4":   // S272, max time T#10S, warning time T#7S
   END_STEP
   TRANSITION ReadOK_3 FROM "Wait reading complete_4" TO DataMove_5   // T287
      := "KeyenceSR1000Ctrl_800A1DB".sHMI.Indata.ReadComplete AND "KeyenceSR1000Ctrl_800A1DB".sHMI.Status.ReadOk;
   END_TRANSITION
   TRANSITION ReadNG_3 FROM "Wait reading complete_4" TO ReadNG3   // T290
      := "KeyenceSR1000Ctrl_800A1DB".sHMI.Status.Complete AND "KeyenceSR1000Ctrl_800A1DB".sHMI.Status.ReadNok;
   END_TRANSITION
   STEP DataMove_6:   // S275, max time T#10S, warning time T#7S
              N    "AutoProcessData".A_Table_1[5].Code:="KeyenceSR1000Ctrl_800A1DB".sHMI.Status.CurrentCode
   END_STEP
   TRANSITION Trans293 FROM DataMove_6 TO "Servo returns to3st Pos_1"   // T295
      := TRUE;
   END_TRANSITION
   STEP ReadNG4:   // S274, max time T#10S, warning time T#7S
          S1  S    "ST10_DeviceError".A.A1TableScan.ScanCodeNG
   END_STEP
   TRANSITION Trans295 FROM ReadNG4 TO "Check reader Ready_5"   // T297, jump
      := #iSysInface.Reset;
   END_TRANSITION
   STEP "Servo returns to4st Pos":   // S18, max time T#10S, warning time T#7S
      interlock C := "ServoV90_A1".Out.oReady;
      (C)     N    "ServoV90_DeviceCtl".V90Servo[1].Point[4].Start
   END_STEP
   TRANSITION Trans19 FROM "Servo returns to4st Pos" TO "Check reader Ready_5"   // T18
      := "ServoV90_DeviceCtl".V90Servo[1].Point[4].Achieve;
   END_TRANSITION
   STEP "Check reader Ready_5":   // S276, max time T#10S, warning time T#7S
   END_STEP
   TRANSITION Trans292 FROM "Check reader Ready_5" TO "Start 4st reading"   // T294
      := "KeyenceSR1000Ctrl_800A1DB".sHMI.Status.Ready;
   END_TRANSITION
   STEP "Wait reading complete_5":   // S278, max time T#10S, warning time T#7S
   END_STEP
   TRANSITION ReadOK_4 FROM "Wait reading complete_5" TO DataMove_6   // T293
      := "KeyenceSR1000Ctrl_800A1DB".sHMI.Indata.ReadComplete AND "KeyenceSR1000Ctrl_800A1DB".sHMI.Status.ReadOk;
   END_TRANSITION
   TRANSITION ReadNG_4 FROM "Wait reading complete_5" TO ReadNG4   // T298
      := "KeyenceSR1000Ctrl_800A1DB".sHMI.Status.Complete AND "KeyenceSR1000Ctrl_800A1DB".sHMI.Status.ReadNok;
   END_TRANSITION
   STEP "Start 4st reading":   // S277, max time T#10S, warning time T#7S
          S1  S    "KeyenceSR1000Ctrl_800A1DB".ioAutoTrigger
   END_STEP
   TRANSITION Trans294 FROM "Start 4st reading" TO "Wait reading complete_5"   // T296
      := NOT "KeyenceSR1000Ctrl_800A1DB".sHMI.Status.Ready;
   END_TRANSITION
   STEP DataMove_1:   // S285, max time T#10S, warning time T#7S
              N    "AutoProcessData".A_Table_1[8].Code:="KeyenceSR1000Ctrl_800A1DB".sHMI.Status.CurrentCode
   END_STEP
   TRANSITION Trans306 FROM DataMove_1 TO "Servo returns to3st Pos_4"   // T329
      := TRUE;
   END_TRANSITION
   STEP ReadNG5:   // S280, max time T#10S, warning time T#7S
          S1  S    "ST10_DeviceError".A.A1TableScan.ScanCodeNG
   END_STEP
   TRANSITION Trans299 FROM ReadNG5 TO "Check reader Ready_6"   // T312, jump
      := #iSysInface.Reset;
   END_TRANSITION
   STEP DataMove_7:   // S281, max time T#10S, warning time T#7S
              N    "AutoProcessData".A_Table_1[6].Code:="KeyenceSR1000Ctrl_800A1DB".sHMI.Status.CurrentCode
   END_STEP
   TRANSITION Trans297 FROM DataMove_7 TO "Servo returns to3st Pos_2"   // T306
      := TRUE;
   END_TRANSITION
   STEP "Servo returns to3st Pos_1":   // S19, max time T#10S, warning time T#7S
      interlock C := "ServoV90_A1".Out.oReady;
      (C)     N    "ServoV90_DeviceCtl".V90Servo[1].Point[5].Start
   END_STEP
   TRANSITION Trans20 FROM "Servo returns to3st Pos_1" TO "Check reader Ready_6"   // T19
      := "ServoV90_DeviceCtl".V90Servo[1].Point[5].Achieve;
   END_TRANSITION
   STEP "Check reader Ready_6":   // S282, max time T#10S, warning time T#7S
   END_STEP
   TRANSITION Trans296 FROM "Check reader Ready_6" TO "Start 5st reading"   // T304
      := "KeyenceSR1000Ctrl_800A1DB".sHMI.Status.Ready;
   END_TRANSITION
   STEP "Start 5st reading":   // S283, max time T#10S, warning time T#7S
          S1  S    "KeyenceSR1000Ctrl_800A1DB".ioAutoTrigger
   END_STEP
   TRANSITION Trans298 FROM "Start 5st reading" TO "Wait reading complete_6"   // T307
      := NOT "KeyenceSR1000Ctrl_800A1DB".sHMI.Status.Ready;
   END_TRANSITION
   STEP "Wait reading complete_6":   // S284, max time T#10S, warning time T#7S
   END_STEP
   TRANSITION ReadOK_5 FROM "Wait reading complete_6" TO DataMove_7   // T299
      := "KeyenceSR1000Ctrl_800A1DB".sHMI.Indata.ReadComplete AND "KeyenceSR1000Ctrl_800A1DB".sHMI.Status.ReadOk;
   END_TRANSITION
   TRANSITION ReadNG_5 FROM "Wait reading complete_6" TO ReadNG5   // T313
      := "KeyenceSR1000Ctrl_800A1DB".sHMI.Status.Complete AND "KeyenceSR1000Ctrl_800A1DB".sHMI.Status.ReadNok;
   END_TRANSITION
   STEP ReadNG7:   // S279, max time T#10S, warning time T#7S
          S1  S    "ST10_DeviceError".A.A1TableScan.ScanCodeNG
   END_STEP
   TRANSITION Trans308 FROM ReadNG7 TO "Check reader Ready_8"   // T337, jump
      := #iSysInface.Reset;
   END_TRANSITION
   STEP ReadNG6:   // S286, max time T#10S, warning time T#7S
          S1  S    "ST10_DeviceError".A.A1TableScan.ScanCodeNG
   END_STEP
   TRANSITION Trans304 FROM ReadNG6 TO "Check reader Ready_7"   // T324, jump
      := #iSysInface.Reset;
   END_TRANSITION
   STEP DataMove_8:   // S287, max time T#10S, warning time T#7S
              N    "AutoProcessData".A_Table_1[7].Code:="KeyenceSR1000Ctrl_800A1DB".sHMI.Status.CurrentCode
   END_STEP
   TRANSITION Trans301 FROM DataMove_8 TO "Servo returns to3st Pos_3"   // T322
      := TRUE;
   END_TRANSITION
   STEP "Servo returns to3st Pos_2":   // S20, max time T#10S, warning time T#7S
      interlock C := "ServoV90_A1".Out.oReady;
      (C)     N    "ServoV90_DeviceCtl".V90Servo[1].Point[6].Start
   END_STEP
   TRANSITION Trans21 FROM "Servo returns to3st Pos_2" TO "Check reader Ready_7"   // T20
      := "ServoV90_DeviceCtl".V90Servo[1].Point[6].Achieve;
   END_TRANSITION
   STEP "Check reader Ready_7":   // S288, max time T#10S, warning time T#7S
   END_STEP
   TRANSITION Trans300 FROM "Check reader Ready_7" TO "Start 6st reading"   // T320
      := "KeyenceSR1000Ctrl_800A1DB".sHMI.Status.Ready;
   END_TRANSITION
   STEP "Start 6st reading":   // S289, max time T#10S, warning time T#7S
          S1  S    "KeyenceSR1000Ctrl_800A1DB".ioAutoTrigger
   END_STEP
   TRANSITION Trans302 FROM "Start 6st reading" TO "Wait reading complete_7"   // T323
      := NOT "KeyenceSR1000Ctrl_800A1DB".sHMI.Status.Ready;
   END_TRANSITION
   STEP "Wait reading complete_7":   // S290, max time T#10S, warning time T#7S
   END_STEP
   TRANSITION ReadOK_6 FROM "Wait reading complete_7" TO DataMove_8   // T315
      := "KeyenceSR1000Ctrl_800A1DB".sHMI.Indata.ReadComplete AND "KeyenceSR1000Ctrl_800A1DB".sHMI.Status.ReadOk;
   END_TRANSITION
   TRANSITION ReadNG_6 FROM "Wait reading complete_7" TO ReadNG6   // T325
      := "KeyenceSR1000Ctrl_800A1DB".sHMI.Status.Complete AND "KeyenceSR1000Ctrl_800A1DB".sHMI.Status.ReadNok;
   END_TRANSITION
   STEP "Servo returns to3st Pos_3":   // S21, max time T#10S, warning time T#7S
      interlock C := "ServoV90_A1".Out.oReady;
      (C)     N    "ServoV90_DeviceCtl".V90Servo[1].Point[7].Start
   END_STEP
   TRANSITION Trans22 FROM "Servo returns to3st Pos_3" TO "Check reader Ready_8"   // T21
      := "ServoV90_DeviceCtl".V90Servo[1].Point[7].Achieve;
   END_TRANSITION
   STEP "Check reader Ready_8":   // S292, max time T#10S, warning time T#7S
   END_STEP
   TRANSITION Trans305 FROM "Check reader Ready_8" TO "Start 7st reading"   // T327
      := "KeyenceSR1000Ctrl_800A1DB".sHMI.Status.Ready;
   END_TRANSITION
   STEP "Start 7st reading":   // S293, max time T#10S, warning time T#7S
          S1  S    "KeyenceSR1000Ctrl_800A1DB".ioAutoTrigger
   END_STEP
   TRANSITION Trans307 FROM "Start 7st reading" TO "Wait reading complete_9"   // T336
      := NOT "KeyenceSR1000Ctrl_800A1DB".sHMI.Status.Ready;
   END_TRANSITION
   STEP "Wait reading complete_9":   // S294, max time T#10S, warning time T#7S
   END_STEP
   TRANSITION ReadOK_7 FROM "Wait reading complete_9" TO DataMove_1   // T326
      := "KeyenceSR1000Ctrl_800A1DB".sHMI.Indata.ReadComplete AND "KeyenceSR1000Ctrl_800A1DB".sHMI.Status.ReadOk;
   END_TRANSITION
   TRANSITION ReadNG_7 FROM "Wait reading complete_9" TO ReadNG7   // T338
      := "KeyenceSR1000Ctrl_800A1DB".sHMI.Status.Complete AND "KeyenceSR1000Ctrl_800A1DB".sHMI.Status.ReadNok;
   END_TRANSITION
   STEP DataMove_2:   // S296, max time T#10S, warning time T#7S
              N    "AutoProcessData".A_Table_1[1].Code:="KeyenceSR1000Ctrl_800A1DB".sHMI.Status.CurrentCode
   END_STEP
   TRANSITION Trans310 FROM DataMove_2 TO Step262   // T348
      := TRUE;
   END_TRANSITION
   STEP ReadNG8:   // S297, max time T#10S, warning time T#7S
          S1  S    "ST10_DeviceError".A.A1TableScan.ScanCodeNG
   END_STEP
   TRANSITION Trans312 FROM ReadNG8 TO "Check reader Ready_9"   // T350, jump
      := #iSysInface.Reset;
   END_TRANSITION
   STEP "Servo returns to3st Pos_4":   // S22, max time T#10S, warning time T#7S
      interlock C := "ServoV90_A1".Out.oReady;
      (C)     N    "ServoV90_DeviceCtl".V90Servo[1].Point[8].Start
   END_STEP
   TRANSITION Trans23 FROM "Servo returns to3st Pos_4" TO "Check reader Ready_9"   // T22
      := "ServoV90_DeviceCtl".V90Servo[1].Point[8].Achieve;
   END_TRANSITION
   STEP "Check reader Ready_9":   // S298, max time T#10S, warning time T#7S
   END_STEP
   TRANSITION Trans309 FROM "Check reader Ready_9" TO "Start 8st reading"   // T346
      := "KeyenceSR1000Ctrl_800A1DB".sHMI.Status.Ready;
   END_TRANSITION
   STEP "Start 8st reading":   // S299, max time T#10S, warning time T#7S
          S1  S    "KeyenceSR1000Ctrl_800A1DB".ioAutoTrigger
   END_STEP
   TRANSITION Trans311 FROM "Start 8st reading" TO "Wait reading complete_10"   // T349
      := NOT "KeyenceSR1000Ctrl_800A1DB".sHMI.Status.Ready;
   END_TRANSITION
   STEP "Wait reading complete_10":   // S304, max time T#10S, warning time T#7S
   END_STEP
   TRANSITION ReadOK_8 FROM "Wait reading complete_10" TO DataMove_2   // T347
      := "KeyenceSR1000Ctrl_800A1DB".sHMI.Indata.ReadComplete AND "KeyenceSR1000Ctrl_800A1DB".sHMI.Status.ReadOk;
   END_TRANSITION
   TRANSITION ReadNG_8 FROM "Wait reading complete_10" TO ReadNG8   // T351
      := "KeyenceSR1000Ctrl_800A1DB".sHMI.Status.Complete AND "KeyenceSR1000Ctrl_800A1DB".sHMI.Status.ReadNok;
   END_TRANSITION
   STEP Step262:   // S306, max time T#10S, warning time T#7S
   END_STEP
   TRANSITION Trans352 FROM Step262 TO CodeCompare   // T352, jump
      := TRUE;
   END_TRANSITION
   STEP "A-Loading-01UpDownTakeCylinderToHP":   // S120, max time T#10S, warning time T#7S
              S    "ST10Cylinder".Cy[2].Inout.AutoGoHome
              R    "ST10Cylinder".Cy[2].Inout.AutoGoWork
   END_STEP
   TRANSITION Trans768 FROM "A-Loading-01UpDownTakeCylinderToHP" TO ReadyReading   // T121
      := NOT "ST10Cylinder".Cy[2].In.WorkPositionSensor AND "ST10Cylinder".Cy[2].In.HomePositionSensor;
   END_TRANSITION
   STEP "A-Loading-01HorizontalCylinderToHP":   // S119, max time T#10S, warning time T#7S
              S    "ST10Cylinder".Cy[1].Inout.AutoGoHome
              R    "ST10Cylinder".Cy[1].Inout.AutoGoWork
   END_STEP
   TRANSITION Trans767 FROM "A-Loading-01HorizontalCylinderToHP" TO ReadyReading   // T120
      := NOT "ST10Cylinder".Cy[1].In.WorkPositionSensor AND "ST10Cylinder".Cy[1].In.HomePositionSensor;
   END_TRANSITION

   // sequencer 4: S200-S299MES查询获取打标数据 / S300-S399 Compare
   STEP CodeCompare:   // S300, max time T#10S, warning time T#7S
   END_STEP
   TRANSITION Trans608 FROM CodeCompare TO Step223   // T608
      := TRUE;
   END_TRANSITION
   STEP 状态刷新100:   // S309, max time T#10S, warning time T#7S
          S1  N    #ioStatus:="MES_CheckIn_OK"
                   //"ST40_IndexTableData_DB".DataOP[1].PublicDta.PartType:="STA10_RecipeActiveDB".ParameterElement.ProcessParameter."M-PartType"
                   //"STA10_ProcessData".Head.PartID:="MEStoPLC_DB".STA10.MainCheckIn."M-PartID"
                   //"ST40_IndexTableData_DB".DataOP[1].PublicDta.RecipeVer:="STA10_RecipeActiveDB".ParameterElement.ProcessParameter."M-RecipeVer"
   END_STEP
   TRANSITION Trans315 FROM 状态刷新100 TO Step400   // T309, jump
      := TRUE;
   END_TRANSITION
   STEP Step223:   // S323, max time T#10S, warning time T#7S
   END_STEP
   TRANSITION Trans235 FROM Step223 TO 状态刷新100   // T335
      := TRUE;
   END_TRANSITION

   // sequencer 5: S400-S499OK&NG数据处理 / S400-S499OK&NG Status Count
   STEP Step400:   // S400, max time T#10S, warning time T#7S
   END_STEP
   TRANSITION Trans224 FROM Step400 TO ProcessFinish   // T400
      := TRUE;
   END_TRANSITION
   STEP ProcessFinish:   // S403, max time T#10S, warning time T#7S
   END_STEP
   TRANSITION Trans405 FROM ProcessFinish TO Step501   // T403, jump
      := TRUE;
   END_TRANSITION

   // sequencer 6: S500-S599 MES上传RFID写入 / S500-S599 MES
   STEP Step501:   // S500, max time T#10S, warning time T#7S
   END_STEP
   TRANSITION Trans407 FROM Step501 TO 准备产品结果数据   // T500
      := TRUE;
   END_TRANSITION
   STEP MES保存开始:   // S503, max time T#10S, warning time T#7S
   END_STEP
   TRANSITION Trans408 FROM MES保存开始 TO 准备产品结果数据_1   // T503
      := (#ioStatus >= "MES_Upload_OK") AND (#ioStatus < "MES_Upload_Complete");
   END_TRANSITION
   TRANSITION Trans419 FROM MES保存开始 TO 数据上传完成   // T520, jump
      := #ioStatus >= "MES_Upload_Complete";
   END_TRANSITION
   STEP 是否在线1:   // S502, max time T#10S, warning time T#7S
   END_STEP
   TRANSITION 在线_1 FROM 是否在线1 TO MES保存开始   // T502
      := "Station_Sys".Cmd.OnOffLine AND NOT "Station_Sys".Cmd.OnOffLine;
   END_TRANSITION
   TRANSITION 离线_1 FROM 是否在线1 TO Step128   // T521
      := NOT "Station_Sys".Cmd.OnOffLine OR "Station_Sys".Cmd.OnOffLine;
   END_TRANSITION
   STEP 准备产品结果数据_1:   // S504, max time T#10S, warning time T#7S
   END_STEP
   TRANSITION Trans27 FROM 准备产品结果数据_1 TO 复位MES保存命令   // T504
      := #准备产品结果数据_1.T > t#100MS;
   END_TRANSITION
   STEP 准备产品结果数据:   // S501, max time T#10S, warning time T#7S
   END_STEP
   TRANSITION Trans26 FROM 准备产品结果数据 TO 是否在线1   // T501
      := #准备产品结果数据.T > t#200MS;
   END_TRANSITION
   STEP 复位MES保存命令:   // S505, max time T#10S, warning time T#7S
              R    "PLCtoMES".Static_2
   END_STEP
   TRANSITION Trans229 FROM 复位MES保存命令 TO "等待MES 保存Ready"   // T505
      := TRUE;
   END_TRANSITION
   STEP 数据上传完成:   // S515, max time T#10S, warning time T#7S
   END_STEP
   TRANSITION Trans619 FROM 数据上传完成 TO "Process Finish"   // T515, jump
      := TRUE;
   END_TRANSITION
   STEP "505准备MES保存数据":   // S507, max time T#10S, warning time T#7S
                   //"Station1UnLoadData".MEStoPLC_CheckOutStation1ST350.PartTypeID:="Station1LoadData".MEStoPLC_CheckInStation1ST350.PartTypeID
                   //"PLCtoMES_DB"."STA10"."MainCheckOut"."P-SubPartID"[1]
                   //"PLCtoMES_DB".STA10.MainCheckOut."P-PartResult":=1
                   //"Station1UnLoadData".MEStoPLC_CheckOutStation1ST350.PartTypeSN:="ST350_RecipeActiveDB".ParameterElement.ProcessParameter."M-RecipeVer"
                   //CALL S_CONV S_CONV
                   //   (IN := "ST350_Sys".TotalCycleTime.No[0]
                   //    OUT => "Station1UnLoadData".MEStoPLC_CheckOutStation1ST350."PLCTransfer time"
                   //     )
              N    #sUpdMES_Data
   END_STEP
   TRANSITION Trans270 FROM "505准备MES保存数据" TO 置位MES保存命令   // T507
      := #"505准备MES保存数据".T > t#100MS;
   END_TRANSITION
   STEP 等待MES保存完成:   // S509, max time T#10S, warning time T#7S
              N    "PLCtoMES".Static_2
   END_STEP
   TRANSITION Trans274 FROM 等待MES保存完成 TO MES保存完成   // T509
      := TRUE;
   END_TRANSITION
   TRANSITION Trans280 FROM 等待MES保存完成 TO "报警 MES保存超时"   // T518
      := #等待MES保存完成.T > t#10S;
   END_TRANSITION
   STEP "等待MES 保存Ready":   // S506, max time T#10S, warning time T#7S
              R    "PLCtoMES".Static_2
   END_STEP
   TRANSITION Trans268 FROM "等待MES 保存Ready" TO "505准备MES保存数据"   // T506
      := NOT "PLCtoMES".Static_2;
   END_TRANSITION
   STEP 等待MES上传复位:   // S511, max time T#10S, warning time T#7S
              R    "PLCtoMES".Static_2
   END_STEP
   TRANSITION Trans605 FROM 等待MES上传复位 TO MES保存结束   // T511
      := TRUE;
   END_TRANSITION
   TRANSITION Trans622 FROM 等待MES上传复位 TO MES上传复位超时   // T516
      := #等待MES上传复位.T > t#10S;
   END_TRANSITION
   STEP 置位MES保存命令:   // S508, max time T#10S, warning time T#7S
   END_STEP
   TRANSITION Trans271 FROM 置位MES保存命令 TO 等待MES保存完成   // T508
      := TRUE;
   END_TRANSITION
   STEP 状态刷新500:   // S514, max time T#10S, warning time T#7S
          S1  N    #ioStatus:=500
   END_STEP
   TRANSITION Trans288 FROM 状态刷新500 TO 数据上传完成   // T514
      := TRUE;
   END_TRANSITION
   STEP "报警 MES保存超时":   // S517, max time T#10S, warning time T#7S
          S1  S    "ST10_DeviceError".MES_Error.CheckInResultOverTime_7
   END_STEP
   TRANSITION Trans281 FROM "报警 MES保存超时" TO 是否在线1   // T519, jump
      := #iSysInface.Reset;
   END_TRANSITION
   STEP MES上传复位超时:   // S516, max time T#10S, warning time T#7S
          S1  S    "ST10_DeviceError".MES_Error.CheckoutCompRstOverTime
   END_STEP
   TRANSITION Trans623 FROM MES上传复位超时 TO 是否在线1   // T517, jump
      := #iSysInface.Reset;
   END_TRANSITION
   STEP MES保存结束:   // S512, max time T#10S, warning time T#7S
   END_STEP
   TRANSITION Trans420 FROM MES保存结束 TO Step617   // T512
      := TRUE;
   END_TRANSITION
   STEP MES保存完成:   // S510, max time T#10S, warning time T#7S
   END_STEP
   TRANSITION Trans624 FROM MES保存完成 TO 等待MES上传复位   // T510
      := #MES保存完成.T > t#500MS;
   END_TRANSITION
   STEP Step617:   // S513, max time T#10S, warning time T#7S
   END_STEP
   TRANSITION Trans255 FROM Step617 TO 状态刷新500   // T513
      := TRUE;
   END_TRANSITION
   STEP Step128:   // S128, max time T#10S, warning time T#7S
   END_STEP
   TRANSITION Trans256 FROM Step128 TO Step617   // T255, jump
      := TRUE;
   END_TRANSITION

   // sequencer 7: S600-S699工件放行 / S600-S699 RobotPick
   STEP "Process Finish":   // S600, max time T#10S, warning time T#7S
              S    #ioPM_Inface.ProcessComplete
              R    #ioPM_Inface.ProcessStart
   END_STEP
   TRANSITION Trans600 FROM "Process Finish" TO CodeCompareResult   // T600
      := TRUE;
   END_TRANSITION
   STEP ProcessFinsh:   // S605, max time T#10S, warning time T#7S: 正式使用时，需要激活复位空循环
   END_STEP
   TRANSITION Trans699 FROM ProcessFinsh TO ProcessStart   // T605, jump
      := TRUE;
   END_TRANSITION
   STEP TableCodeReady:   // S307, max time T#10S, warning time T#7S
   END_STEP
   TRANSITION Trans290 FROM TableCodeReady TO WaitFixtureScanFinish   // T604
      := TRUE;
   END_TRANSITION
   STEP CodeCompareResult:   // S308, max time T#10S, warning time T#7S
   END_STEP
   TRANSITION Trans609 FROM CodeCompareResult TO TableCodeReady   // T609
      := "AutoProcessData".GlobalData.Table1CodeOKFlag AND (#CodeCompareResult.T > t#100MS);
   END_TRANSITION
   TRANSITION Trans610 FROM CodeCompareResult TO "Barcode mismatch"   // T610
      := NOT "AutoProcessData".GlobalData.Table1CodeOKFlag AND (#CodeCompareResult.T > t#100MS);
   END_TRANSITION
   STEP WaitChangeOverFinish:   // S310, max time T#10S, warning time T#7S
   END_STEP
   TRANSITION Trans611 FROM WaitChangeOverFinish TO WaitChangeOverStart   // T611
      := "ChangeOver_DB".Global.AllFixtureScanCompareOk;
   END_TRANSITION
   TRANSITION Trans617 FROM WaitChangeOverFinish TO ProcessFinsh   // T616
      := "ChangeOver_DB".Global.ScanFixtureFlag;
   END_TRANSITION
   STEP WaitChangeOverStart:   // S312, max time T#10S, warning time T#7S
   END_STEP
   TRANSITION Trans612 FROM WaitChangeOverStart TO ProcessFinsh   // T612
      := NOT "ChangeOver_DB".Global.AllFixtureScanCompareOk;
   END_TRANSITION
   STEP "Barcode mismatch":   // S313, max time T#10S, warning time T#7S
   END_STEP
   TRANSITION Trans614 FROM "Barcode mismatch" TO ProcessStart   // T613, jump
      := #iSysInface.Reset;
   END_TRANSITION
   STEP WaitFixtureScanFinish:   // S314, max time T#10S, warning time T#7S
   END_STEP
   TRANSITION Trans616 FROM WaitFixtureScanFinish TO WaitChangeOverFinish   // T615
      := NOT "ChangeOver_DB".Global.ScanFixtureFlag;
   END_TRANSITION

   // permanent post-instructions
   NETWORK 1
      #ioPM_Inface.StepNum := #RT_DATA.S_DISPLAY;
   NETWORK 2
      IF #iSysInface.Reset THEN #AlarmID := 0; END_IF;
   NETWORK 3
      #TON[10].TON(IN := #工件放行中, PT := T#0.5S);
      IF #TON[10].Q THEN #工件放行中 := FALSE; END_IF;
END_FUNCTION_BLOCK

FUNCTION_BLOCK "SysFlowCtrlGraph"   // FB3006, SCL
{ S7_Optimized_Access := 'TRUE' }
// stored: AutoNumber false, MemoryReserve 100, SetENOAutomatically false
   VAR_INPUT
      INIT : Bool;
      iSysInface : "RCS_SysComInterface_V1";
   END_VAR
   VAR_IN_OUT
      ioPM_Inface : "RCS_PMInterface_V1";
      ioGraphCtrl : G7_MOPPlus_V6;
   END_VAR
   VAR
      sHis : Array[0..7] of Bool;
      sSetInitialDelay : TON_TIME;
      S_NEXT_Delay { S7_SetPoint := 'True'} : Array[0..1] of TON_TIME;
   END_VAR
BEGIN
   (*############################################################
      RUHLAMAT SUZHOU ELEC.STD.
      Copyright (c) 2022. All rights reserved.    

      NAME OF FUNCTION BLOCK:         SysFlowCtrlGraph
      VERSION NUMBER:                 V1.0
      COMPOSER:                       Ming.Jiang

      LAST CHANGE:                    1.Dece.2022
      Comment by Ming.Jiang 

      #RET_VALUE:


      #Alert Value:


      -----------------------------------------------------
      Date        Name      Version           Activity                                                                              

   ############################################################*)

   REGION Control Mode
       //AUTO:Auto Mode
       #ioGraphCtrl.AUTO := #ioGraphCtrl.SUP := #iSysInface.Auto.Mode;

       //MAN:Manual Mode
       #ioGraphCtrl.MAN :=  #iSysInface.ManualMode;
       #ioGraphCtrl.OFF := #ioPM_Inface.AlarmImdilyStop OR #iSysInface.ManualMode;
       IF #iSysInface.ManualMode OR #ioPM_Inface.AlarmImdilyStop THEN
           #ioPM_Inface.InitialRun      := 0;
           #ioPM_Inface.InitialOK       := 0;
           #ioPM_Inface.WaitRunning     := 0;
           // #ioPM_Inface.Running         := 0;
           #ioPM_Inface.UnPause    := 0;
           #ioPM_Inface.ProcessComplete := 0;

       END_IF;
       //AutoRunning
       //
       // #ioPM_Inface.Running := ((#iSysInface.Auto.StartAuto AND #iSysInface.Ready) OR #iSysInface.Auto.Running)
       // AND AND NOT "ST10_Sys".Auto.RunningOver 

       IF NOT #iSysInface.ManualMode AND #iSysInface.SysRun AND #ioPM_Inface.InitialOK AND NOT #ioPM_Inface.Alarm
           AND NOT #ioPM_Inface.AlarmImdilyStop AND NOT #iSysInface.Auto.RunningPause THEN
           IF #iSysInface.Auto.StartAuto AND #iSysInface.Ready AND  NOT  #ioPM_Inface.Running  THEN
               #ioPM_Inface.Running := 1;
           END_IF;
       ELSE
           #ioPM_Inface.Running := 0;
       END_IF;

       //Step Num






       //TAP:StepMode
       #ioGraphCtrl.TAP := #iSysInface.Auto.StepMode;
       #ioGraphCtrl.T_PUSH := #iSysInface.Auto.StepMode AND #ioPM_Inface.SetNextStep AND NOT #sHis[0];
       #sHis[0] := #ioPM_Inface.SetNextStep;

       //INTERLOCK
       #ioGraphCtrl.LOCK    := 1;
       #ioGraphCtrl.IL_PERM := 1;
       #ioGraphCtrl.T_PERM  := 1;

   END_REGION

   REGION Initialization

     #sSetInitialDelay(IN := #iSysInface.SetInitial OR #ioPM_Inface.SetInitial OR #INIT,
                         PT := T#2000ms);//20221221DB

       IF #sSetInitialDelay.Q AND #iSysInface.SysRun AND NOT #iSysInface.ManualMode THEN

           IF NOT #sHis[1] THEN
               //     #oStatus.Initializing := TRUE;
               //     #oStatus.InitializeOK := 0;
               //     #oStatus.WaitRunning := 0;
               //     #oStatus.Running := 0;
               //     #oStatus.RunningPause := 0;
               //     #oStatus.RunningFinished := 0;
               #ioGraphCtrl.INIT := #sSetInitialDelay.Q;
           END_IF;

       ELSE
           #ioGraphCtrl.INIT := 0;
       END_IF;
       #sHis[1] := #sSetInitialDelay.Q;
   END_REGION

   REGION Reset
       //
       #ioGraphCtrl.ACK := #iSysInface.Reset;


   END_REGION

   REGION Running and Pause(Halt)
       #ioGraphCtrl.HALT :=(#ioPM_Inface.InitialOK AND NOT #ioPM_Inface.Running )  OR   #ioPM_Inface.Alarm OR #ioPM_Inface.AlarmImdilyStop ; //#ioPM_Inface.UnPause  NOT #iSysInface.Auto.RunningPause
       #ioGraphCtrl.OPS_ZERO := #iSysInface.ManualMode OR NOT #iSysInface.SysRun OR #ioPM_Inface.AlarmImdilyStop ;
       #ioGraphCtrl.TMS_HALT := #iSysInface.ManualMode OR NOT #iSysInface.SysRun OR #ioPM_Inface.AlarmImdilyStop;
   END_REGION


   #S_NEXT_Delay[0](PT := t#3s,
                 IN := #ioGraphCtrl.S_NEXT);

   IF #S_NEXT_Delay[0].Q THEN
       #ioGraphCtrl.S_NEXT := 0;

   END_IF;

   #S_NEXT_Delay[1](PT := t#3s,
                    IN := NOT #ioGraphCtrl.S_NEXT);

   IF #S_NEXT_Delay[1].Q THEN
       #ioGraphCtrl.S_NEXT := 1;
   END_IF;
END_FUNCTION_BLOCK

FUNCTION_BLOCK "ST10_Flow2_A1TableUnloading"   // FB1072, GRAPH
// stored: AcknowledgeErrorsRequired false, AutoNumber false, GraphVersion 6.0, InitialValuesAcquisition false, SetENOAutomatically false
   // inherited from GRAPH_BASE
   VAR_INPUT
      iSysInface : "RCS_SysComInterface_V1";
   END_VAR
   VAR_IN_OUT
      ioPM_Inface : "RCS_PMInterface_V1";
      ioStatus : Int;
   END_VAR
   VAR
      sCtrlMode { S7_SetPoint := 'True'} : "SysFlowCtrlGraph";
      sUpdMES_Data : Bool;   // 更新MES数据
      工件放行中 : Bool;
      前站站号 { ExternalAccessible := 'False'; ExternalVisible := 'False'; ExternalWritable := 'False'} : UInt;
      本站站号 { ExternalAccessible := 'False'; ExternalVisible := 'False'; ExternalWritable := 'False'} : UInt;
      弹窗Temp : Array[1..10] of Int;
      AlarmID : Int;
      TON { S7_SetPoint := 'True'} : Array[0..10] of TON_TIME;
      TOF { S7_SetPoint := 'True'} : Array[0..10] of TOF_TIME;
      sUP { S7_SetPoint := 'True'} : Array[0..10] of Bool;
      更新RFID完成 : Bool;
   END_VAR
   VAR_TEMP
      Tempresult : USInt;
      本站站号乘10 : UInt;
   END_VAR
   // // TON[0] : 托盘流入1托盘到位传感器 / iA-Rotating product Check
   // // TON[1] : 托盘流入1托盘到位传感器
   // // TON[2] : 托盘流入1产品有无传感器
   // // TON[3] : 托盘流入1产品有无传感器
   // // TON[4] : 托盘流入1姿态检测光电2
   // // TON[5] : 托盘流入1姿态检测光电3
   // // TON[0].Q : 托盘流入1托盘到位 / iA-Rotating product Check
   // // TON[1].Q : 托盘流入1托盘无
   // // TON[2].Q : 托盘流入1有产品
   // // TON[3].Q : 托盘流入1无产品
   // // TON[4].Q : 托盘流入1姿态检测光电2
   // // TON[5].Q : 托盘流入1姿态检测光电3
   // // TOF[1] : iA-Rotating product Check
BEGIN
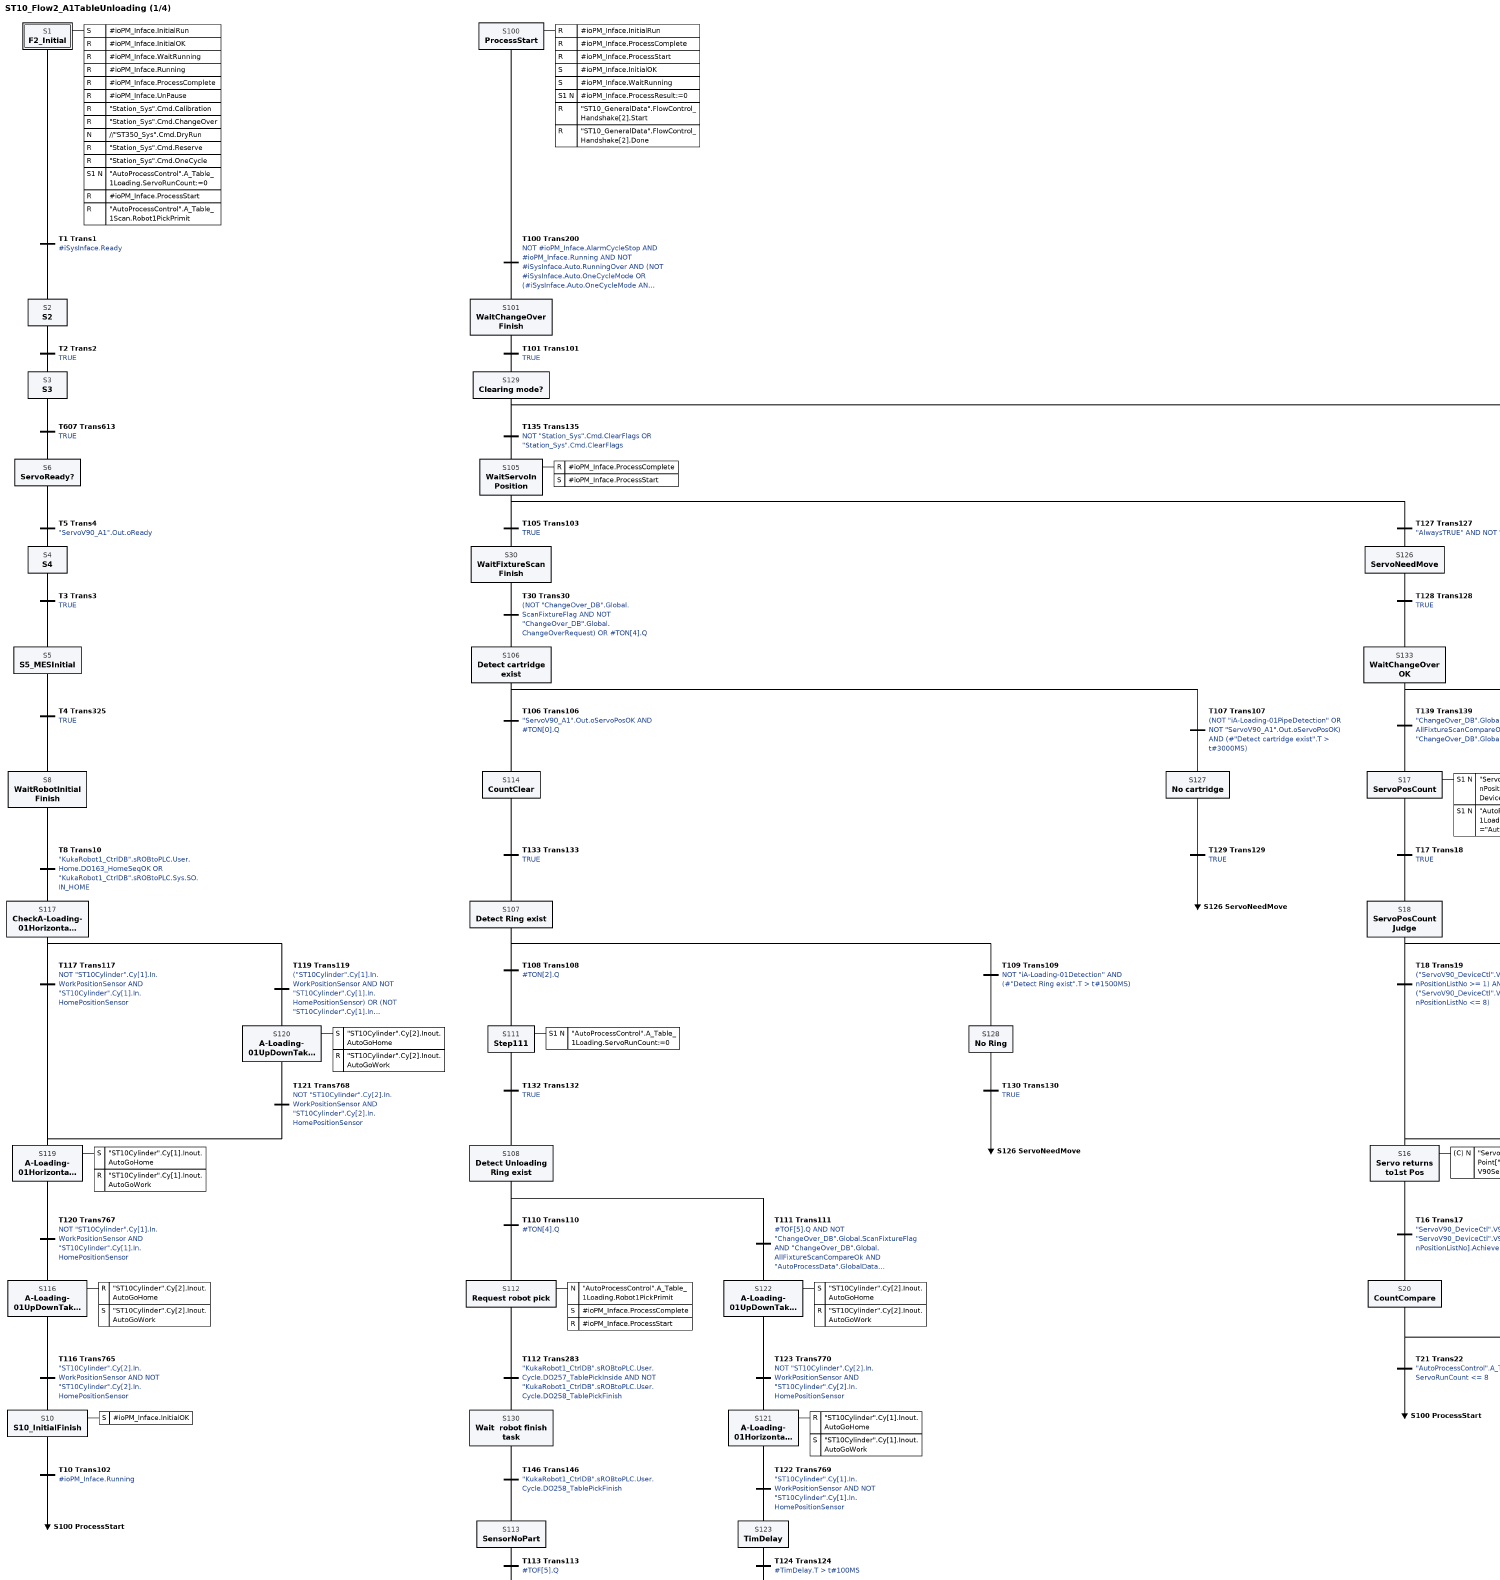
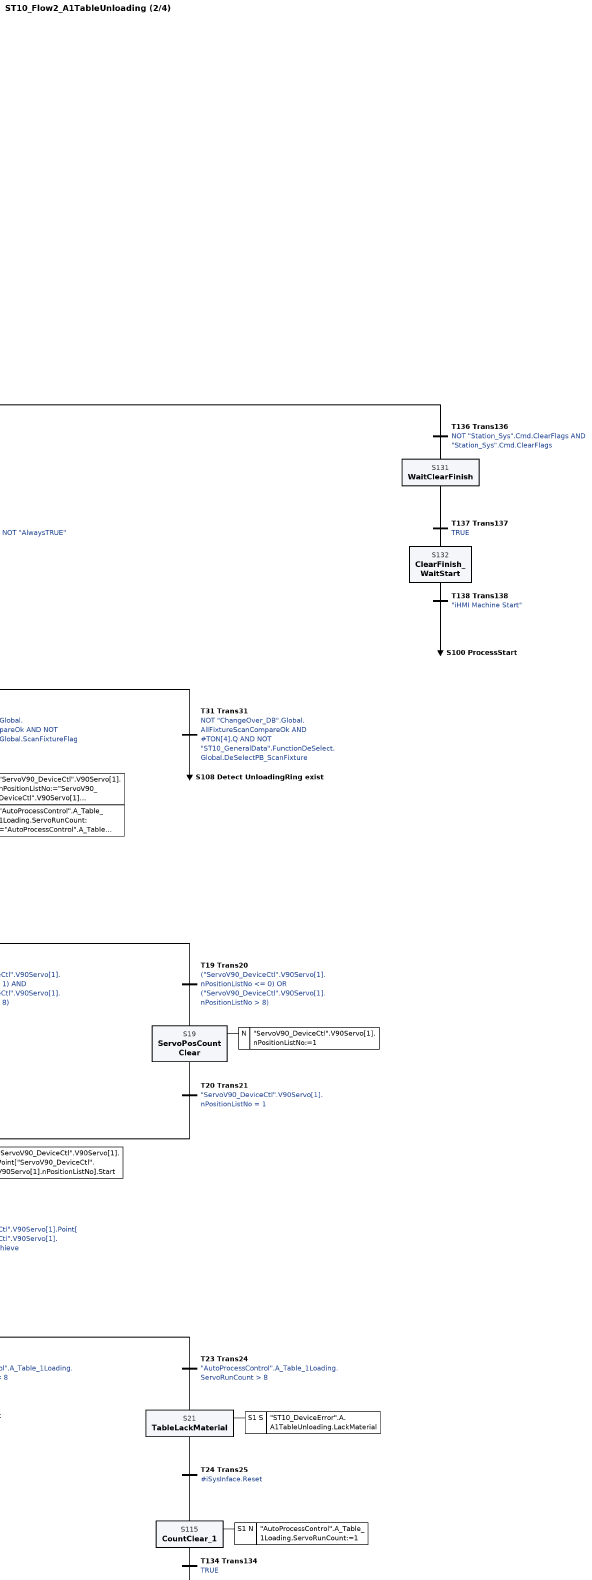
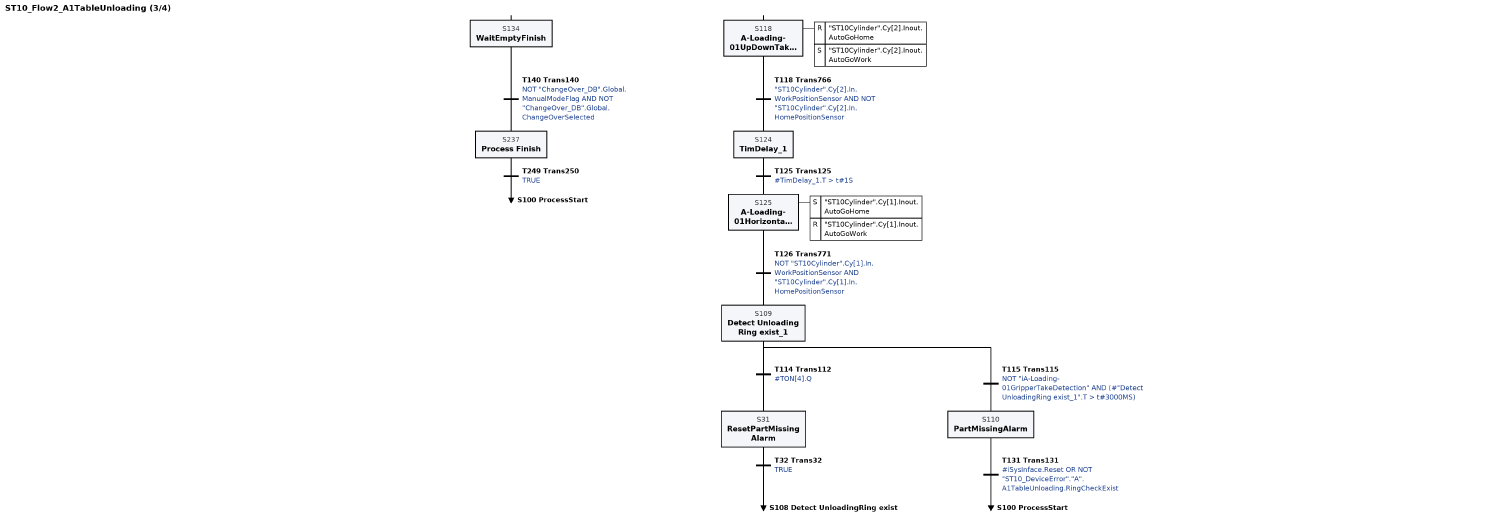
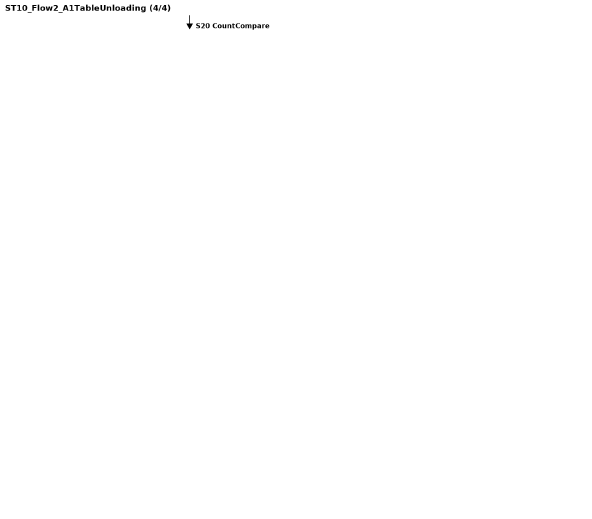
   // permanent pre-instructions
   NETWORK 1
      #TON[10].TON(IN := "AlwaysTRUE" AND "Station_Sys".Alarm.ImmediatelyStop, PT := T#300ms);
      #ioPM_Inface.AlarmImdilyStop := #TON[10].Q;
      #ioPM_Inface.AlarmCycleStop := "AlwaysTRUE" AND "Station_Sys".Alarm.CycleStop;
   NETWORK 2
      IF NOT False THEN
          #sCtrlMode(iSysInface := #iSysInface, ioPM_Inface := #ioPM_Inface, ioGraphCtrl := #RT_DATA.MOP);   // "SysFlowCtrlGraph"
      END_IF;
   NETWORK 3
      #TON[0].TON(IN := "AlwaysTRUE" AND "iA-Loading-01PipeDetection", PT := t#500ms);   // 工位11有托盘
      #TOF[1].TOF(IN := "AlwaysTRUE" AND NOT "iA-Loading-01PipeDetection", PT := T#300ms);   // 工位无托盘
      #TON[2].TON(IN := "AlwaysTRUE" AND "iA-Loading-01Detection", PT := T#300ms);
      #TOF[3].TOF(IN := "AlwaysTRUE" AND NOT "iA-Loading-01Detection", PT := T#300ms);
      #TON[4].TON(IN := "AlwaysTRUE" AND "iA-Loading-01GripperTakeDetection", PT := T#300ms);
      #TOF[5].TOF(IN := "AlwaysTRUE" AND NOT "iA-Loading-01GripperTakeDetection", PT := T#300ms);
   NETWORK 4
      #前站站号 := 345;
      #本站站号 := 350;

   // sequencer 1: S01-S99 初始化 / S01-S99 Initial
   INITIAL_STEP F2_Initial:   // S1, max time T#10S, warning time T#7S
              S    #ioPM_Inface.InitialRun
              R    #ioPM_Inface.InitialOK
              R    #ioPM_Inface.WaitRunning
              R    #ioPM_Inface.Running
              R    #ioPM_Inface.ProcessComplete
              R    #ioPM_Inface.UnPause
              R    "Station_Sys".Cmd.Calibration
              R    "Station_Sys".Cmd.ChangeOver
                   //"ST350_Sys".Cmd.DryRun
              R    "Station_Sys".Cmd.Reserve
              R    "Station_Sys".Cmd.OneCycle
          S1  N    "AutoProcessControl".A_Table_1Loading.ServoRunCount:=0
              R    #ioPM_Inface.ProcessStart
              R    "AutoProcessControl".A_Table_1Scan.Robot1PickPrimit
              R    "AutoProcessControl".A_Table_1Loading.Robot1PickPrimit
              R    "AutoProcessControl".A_Table_2Scan.Robot3PickPrimit
              R    "AutoProcessControl".A_Table_2Loading.Robot3PickPrimit
              R    "AutoProcessControl".A_ScanRotary.Robot1PickPrimit
              R    "AutoProcessControl".A_ScanRotary.Robot1PutPrimit
              R    "AutoProcessControl".H_ShafeLine.Robot1PickPrimit
              R    "AutoProcessControl".J_MagnetLine.Robot2PickPrimit
              R    "AutoProcessControl".K_ShafeLine.Robot2PickPrimit
              R    "AutoProcessControl".L_ShafeLine.Robot3PutPrimit
   END_STEP
   TRANSITION Trans1 FROM F2_Initial TO S2   // T1
      := #iSysInface.Ready;
   END_TRANSITION
   STEP S2:   // S2, max time T#10S, warning time T#7S
   END_STEP
   TRANSITION Trans2 FROM S2 TO S3   // T2
      := TRUE;
   END_TRANSITION
   STEP S4:   // S4, max time T#10S, warning time T#7S
   END_STEP
   TRANSITION Trans3 FROM S4 TO S5_MESInitial   // T3
      := TRUE;
   END_TRANSITION
   STEP S5_MESInitial:   // S5, max time T#10S, warning time T#7S
   END_STEP
   TRANSITION Trans325 FROM S5_MESInitial TO WaitRobotInitialFinish   // T4
      := TRUE;
   END_TRANSITION
   STEP S10_InitialFinish:   // S10, max time T#10S, warning time T#7S
              S    #ioPM_Inface.InitialOK
   END_STEP
   TRANSITION Trans102 FROM S10_InitialFinish TO ProcessStart   // T10, jump
      := #ioPM_Inface.Running;
   END_TRANSITION
   STEP S3:   // S3, max time T#10S, warning time T#7S
   END_STEP
   TRANSITION Trans613 FROM S3 TO "ServoReady?"   // T607
      := TRUE;
   END_TRANSITION
   STEP WaitRobotInitialFinish:   // S8, max time T#10S, warning time T#7S
   END_STEP
   TRANSITION Trans10 FROM WaitRobotInitialFinish TO "CheckA-Loading-01HorizontalCylindePos"   // T8
      := "KukaRobot1_CtrlDB".sROBtoPLC.User.Home.DO163_HomeSeqOK OR "KukaRobot1_CtrlDB".sROBtoPLC.Sys.SO.IN_HOME;
   END_TRANSITION
   STEP "A-Loading-01UpDownTakeCylinderToHP_2":   // S120, max time T#10S, warning time T#7S
              S    "ST10Cylinder".Cy[2].Inout.AutoGoHome
              R    "ST10Cylinder".Cy[2].Inout.AutoGoWork
   END_STEP
   TRANSITION Trans768 FROM "A-Loading-01UpDownTakeCylinderToHP_2" TO "A-Loading-01HorizontalCylinderToHP"   // T121
      := NOT "ST10Cylinder".Cy[2].In.WorkPositionSensor AND "ST10Cylinder".Cy[2].In.HomePositionSensor;
   END_TRANSITION
   STEP "CheckA-Loading-01HorizontalCylindePos":   // S117, max time T#10S, warning time T#7S
   END_STEP
   TRANSITION Trans117 FROM "CheckA-Loading-01HorizontalCylindePos" TO "A-Loading-01HorizontalCylinderToHP"   // T117
      := NOT "ST10Cylinder".Cy[1].In.WorkPositionSensor AND "ST10Cylinder".Cy[1].In.HomePositionSensor;
   END_TRANSITION
   TRANSITION Trans119 FROM "CheckA-Loading-01HorizontalCylindePos" TO "A-Loading-01UpDownTakeCylinderToHP_2"   // T119
      := ("ST10Cylinder".Cy[1].In.WorkPositionSensor AND NOT "ST10Cylinder".Cy[1].In.HomePositionSensor) OR (NOT "ST10Cylinder".Cy[1].In.WorkPositionSensor AND NOT "ST10Cylinder".Cy[1].In.HomePositionSensor);
   END_TRANSITION
   STEP "A-Loading-01HorizontalCylinderToHP":   // S119, max time T#10S, warning time T#7S
              S    "ST10Cylinder".Cy[1].Inout.AutoGoHome
              R    "ST10Cylinder".Cy[1].Inout.AutoGoWork
   END_STEP
   TRANSITION Trans767 FROM "A-Loading-01HorizontalCylinderToHP" TO "A-Loading-01UpDownTakeCylinderToWP"   // T120
      := NOT "ST10Cylinder".Cy[1].In.WorkPositionSensor AND "ST10Cylinder".Cy[1].In.HomePositionSensor;
   END_TRANSITION
   STEP "A-Loading-01UpDownTakeCylinderToWP":   // S116, max time T#10S, warning time T#7S
              R    "ST10Cylinder".Cy[2].Inout.AutoGoHome
              S    "ST10Cylinder".Cy[2].Inout.AutoGoWork
   END_STEP
   TRANSITION Trans765 FROM "A-Loading-01UpDownTakeCylinderToWP" TO S10_InitialFinish   // T116
      := "ST10Cylinder".Cy[2].In.WorkPositionSensor AND NOT "ST10Cylinder".Cy[2].In.HomePositionSensor;
   END_TRANSITION
   STEP "ServoReady?":   // S6, max time T#10S, warning time T#7S
   END_STEP
   TRANSITION Trans4 FROM "ServoReady?" TO S4   // T5
      := "ServoV90_A1".Out.oReady;
   END_TRANSITION

